LIN {X 0,Y 260.173,Z 449.996,A -85,B 0,C 180,E1 11651.487,E2 11651.487} C_VEL
LIN {X 0,Y 247.956,Z 426.22,A -85,B 0,C 180,E1 11648.205,E2 11648.205} C_VEL
LIN {X 0,Y 243.469,Z 417.822,A -85,B 0,C 180,E1 11646.84,E2 11646.84} C_VEL
LIN {X 0,Y 237.54,Z 404.393,A -85,B 0,C 180,E1 11643.464,E2 11643.464} C_VEL
LIN {X 0,Y 234.75,Z 397.683,A -85,B 0,C 180,E1 11641.737,E2 11641.737} C_VEL
LIN {X 0,Y 234.741,Z 397.554,A -85,B 0,C 180,E1 11636.558,E2 11636.558} C_VEL
LIN {X 0,Y 234.73,Z 397.556,A -85,B 0,C 180,E1 11631.489,E2 11631.489} C_VEL
LIN {X 0,Y 234.745,Z 397.554,A -85,B 0,C 180,E1 11626.327,E2 11626.327} C_VEL
LIN {X 0,Y 234.727,Z 397.561,A -85,B 0,C 180,E1 11621.3,E2 11621.3} C_VEL
LIN {X 0,Y 234.75,Z 397.558,A -85,B 0,C 180,E1 11616.113,E2 11616.113} C_VEL
LIN {X 0,Y 234.722,Z 397.559,A -85,B 0,C 180,E1 11610.976,E2 11610.976} C_VEL
LIN {X 0,Y 234.739,Z 397.555,A -85,B 0,C 180,E1 11605.847,E2 11605.847} C_VEL
LIN {X 0,Y 234.724,Z 397.557,A -85,B 0,C 180,E1 11600.685,E2 11600.685} C_VEL
LIN {X 0,Y 234.752,Z 397.559,A -85,B 0,C 180,E1 11595.698,E2 11595.698} C_VEL
LIN {X 0,Y 234.734,Z 397.56,A -85,B 0,C 180,E1 11590.282,E2 11590.282} C_VEL
LIN {X 0,Y 234.736,Z 397.556,A -85,B 0,C 180,E1 11585.327,E2 11585.327} C_VEL
LIN {X 0,Y 234.735,Z 397.557,A -85,B 0,C 180,E1 11580.108,E2 11580.108} C_VEL
LIN {X 0,Y 234.732,Z 397.564,A -85,B 0,C 180,E1 11575.195,E2 11575.195} C_VEL
LIN {X 0,Y 234.756,Z 397.673,A -85,B 0,C 180,E1 11573.699,E2 11573.699} C_VEL
LIN {X 0,Y 239.266,Z 412.086,A -85,B 0,C 180,E1 11568.68,E2 11568.68} C_VEL
LIN {X 0,Y 243.442,Z 426.646,A -85,B 0,C 180,E1 11564.048,E2 11564.048} C_VEL
LIN {X 0,Y 247.26,Z 441.444,A -85,B 0,C 180,E1 11559.711,E2 11559.711} C_VEL
LIN {X 0,Y 250.149,Z 453.996,A -85,B 0,C 180,E1 11556.269,E2 11556.269} C_VEL
LIN {X 0,Y 245.768,Z 476.519,A -85,B 0,C 180,E1 11551.382,E2 11551.382} C_VEL
LIN {X 0,Y 248.92,Z 517.799,A -85,B 0,C 180,E1 11548.969,E2 11548.969} C_VEL
LIN {X 0,Y 248.866,Z 523.548,A -85,B 0,C 180,E1 11548.677,E2 11548.677} C_VEL
LIN {X 0,Y 242.887,Z 615.376,A -85,B 0,C 180,E1 11544.277,E2 11544.277} C_VEL
LIN {X 0,Y 241.688,Z 633.773,A -85,B 0,C 180,E1 11542.949,E2 11542.949} C_VEL
LIN {X 0,Y 240.184,Z 651.793,A -85,B 0,C 180,E1 11541.173,E2 11541.173} C_VEL
LIN {X 0,Y 238.661,Z 668.194,A -85,B 0,C 180,E1 11539.074,E2 11539.074} C_VEL
LIN {X 0,Y 238.095,Z 674.333,A -85,B 0,C 180,E1 11538.142,E2 11538.142} C_VEL
LIN {X 0,Y 236.506,Z 680.701,A -85,B 0,C 180,E1 11537.118,E2 11537.118} C_VEL
LIN {X 0,Y 230.234,Z 693.25,A -85,B 0,C 180,E1 11534.856,E2 11534.856} C_VEL
LIN {X 0,Y 227.886,Z 699.683,A -85,B 0,C 180,E1 11533.431,E2 11533.431} C_VEL
LIN {X 0,Y 227.659,Z 701.248,A -85,B 0,C 180,E1 11533.044,E2 11533.044} C_VEL
LIN {X 0,Y 226.821,Z 712.8,A -85,B 0,C 180,E1 11529.9,E2 11529.9} C_VEL
LIN {X 0,Y 226.363,Z 723.238,A -85,B 0,C 180,E1 11526.34,E2 11526.34} C_VEL
LIN {X 0,Y 226.411,Z 731.344,A -85,B 0,C 180,E1 11522.785,E2 11522.785} C_VEL
LIN {X 0,Y 227.03,Z 738.033,A -85,B 0,C 180,E1 11518.991,E2 11518.991} C_VEL
LIN {X 0,Y 228.408,Z 742.937,A -85,B 0,C 180,E1 11514.978,E2 11514.978} C_VEL
LIN {X 0,Y 230.514,Z 745.783,A -85,B 0,C 180,E1 11511.268,E2 11511.268} C_VEL
LIN {X 0,Y 233.668,Z 746.873,A -85,B 0,C 180,E1 11507.395,E2 11507.395} C_VEL
LIN {X 0,Y 237.813,Z 746.163,A -85,B 0,C 180,E1 11503.639,E2 11503.639} C_VEL
LIN {X 0,Y 242.935,Z 743.576,A -85,B 0,C 180,E1 11500.025,E2 11500.025} C_VEL
LIN {X 0,Y 249.037,Z 739.206,A -85,B 0,C 180,E1 11496.58,E2 11496.58} C_VEL
LIN {X 0,Y 255.625,Z 733.401,A -85,B 0,C 180,E1 11493.519,E2 11493.519} C_VEL
LIN {X 0,Y 264.087,Z 724.771,A -85,B 0,C 180,E1 11490.266,E2 11490.266} C_VEL
LIN {X 0,Y 272.968,Z 714.412,A -85,B 0,C 180,E1 11487.422,E2 11487.422} C_VEL
LIN {X 0,Y 281.754,Z 702.992,A -85,B 0,C 180,E1 11485.06,E2 11485.06} C_VEL
LIN {X 0,Y 291.09,Z 689.414,A -85,B 0,C 180,E1 11482.928,E2 11482.928} C_VEL
LIN {X 0,Y 299.888,Z 674.728,A -85,B 0,C 180,E1 11481.185,E2 11481.185} C_VEL
LIN {X 0,Y 304.796,Z 665.496,A -85,B 0,C 180,E1 11480.292,E2 11480.292} C_VEL
LIN {X 0,Y 295.693,Z 684.166,A -85,B 0,C 180,E1 11479.091,E2 11479.091} C_VEL
LIN {X 0,Y 286.363,Z 701.007,A -85,B 0,C 180,E1 11477.602,E2 11477.602} C_VEL
LIN {X 0,Y 276.278,Z 717.417,A -85,B 0,C 180,E1 11475.624,E2 11475.624} C_VEL
LIN {X 0,Y 266.118,Z 732.842,A -85,B 0,C 180,E1 11473.142,E2 11473.142} C_VEL
LIN {X 0,Y 256.713,Z 746.406,A -85,B 0,C 180,E1 11470.282,E2 11470.282} C_VEL
LIN {X 0,Y 247.986,Z 758.698,A -85,B 0,C 180,E1 11466.924,E2 11466.924} C_VEL
LIN {X 0,Y 240.245,Z 769.768,A -85,B 0,C 180,E1 11463.039,E2 11463.039} C_VEL
LIN {X 0,Y 233.52,Z 779.982,A -85,B 0,C 180,E1 11458.377,E2 11458.377} C_VEL
LIN {X 0,Y 228.844,Z 788.193,A -85,B 0,C 180,E1 11453.428,E2 11453.428} C_VEL
LIN {X 0,Y 226.352,Z 794.238,A -85,B 0,C 180,E1 11448.545,E2 11448.545} C_VEL
LIN {X 0,Y 225.176,Z 804.136,A -85,B 0,C 180,E1 11444.398,E2 11444.398} C_VEL
LIN {X 0,Y 224.691,Z 811.895,A -85,B 0,C 180,E1 11440.253,E2 11440.253} C_VEL
LIN {X 0,Y 224.74,Z 817.761,A -85,B 0,C 180,E1 11436.13,E2 11436.13} C_VEL
LIN {X 0,Y 224.855,Z 821.641,A -85,B 0,C 180,E1 11432.294,E2 11432.294} C_VEL
LIN {X 0,Y 224.745,Z 823.926,A -85,B 0,C 180,E1 11428.725,E2 11428.725} C_VEL
LIN {X 0,Y 224.369,Z 825.073,A -85,B 0,C 180,E1 11424.63,E2 11424.63} C_VEL
LIN {X 0,Y 224.279,Z 824.752,A -85,B 0,C 180,E1 11419.987,E2 11419.987} C_VEL
LIN {X 0,Y 225.314,Z 822.532,A -85,B 0,C 180,E1 11414.822,E2 11414.822} C_VEL
LIN {X 0,Y 228.103,Z 818.227,A -85,B 0,C 180,E1 11409.472,E2 11409.472} C_VEL
LIN {X 0,Y 232.879,Z 811.96,A -85,B 0,C 180,E1 11404.301,E2 11404.301} C_VEL
LIN {X 0,Y 239.69,Z 803.753,A -85,B 0,C 180,E1 11399.408,E2 11399.408} C_VEL
LIN {X 0,Y 248.538,Z 793.638,A -85,B 0,C 180,E1 11394.88,E2 11394.88} C_VEL
LIN {X 0,Y 259.353,Z 781.523,A -85,B 0,C 180,E1 11390.783,E2 11390.783} C_VEL
LIN {X 0,Y 271.422,Z 768.109,A -85,B 0,C 180,E1 11387.327,E2 11387.327} C_VEL
LIN {X 0,Y 284.436,Z 753.541,A -85,B 0,C 180,E1 11384.472,E2 11384.472} C_VEL
LIN {X 0,Y 288.888,Z 748.523,A -85,B 0,C 180,E1 11383.627,E2 11383.627} C_VEL
LIN {X 0,Y 276.067,Z 761.536,A -85,B 0,C 180,E1 11380.687,E2 11380.687} C_VEL
LIN {X 0,Y 264.26,Z 772.98,A -85,B 0,C 180,E1 11377.256,E2 11377.256} C_VEL
LIN {X 0,Y 253.496,Z 782.998,A -85,B 0,C 180,E1 11373.247,E2 11373.247} C_VEL
LIN {X 0,Y 244.427,Z 790.978,A -85,B 0,C 180,E1 11368.861,E2 11368.861} C_VEL
LIN {X 0,Y 237.116,Z 796.985,A -85,B 0,C 180,E1 11364.143,E2 11364.143} C_VEL
LIN {X 0,Y 231.58,Z 801.07,A -85,B 0,C 180,E1 11359.155,E2 11359.155} C_VEL
LIN {X 0,Y 227.872,Z 803.179,A -85,B 0,C 180,E1 11354.137,E2 11354.137} C_VEL
LIN {X 0,Y 225.685,Z 803.454,A -85,B 0,C 180,E1 11349.177,E2 11349.177} C_VEL
LIN {X 0,Y 224.64,Z 801.992,A -85,B 0,C 180,E1 11344.339,E2 11344.339} C_VEL
LIN {X 0,Y 224.296,Z 798.959,A -85,B 0,C 180,E1 11339.744,E2 11339.744} C_VEL
LIN {X 0,Y 224.27,Z 794.49,A -85,B 0,C 180,E1 11335.397,E2 11335.397} C_VEL
LIN {X 0,Y 224.606,Z 788.308,A -85,B 0,C 180,E1 11331.036,E2 11331.036} C_VEL
LIN {X 0,Y 225.458,Z 780.224,A -85,B 0,C 180,E1 11326.667,E2 11326.667} C_VEL
LIN {X 0,Y 226.903,Z 770.573,A -85,B 0,C 180,E1 11322.563,E2 11322.563} C_VEL
LIN {X 0,Y 228.921,Z 759.495,A -85,B 0,C 180,E1 11318.745,E2 11318.745} C_VEL
LIN {X 0,Y 231.574,Z 746.383,A -85,B 0,C 180,E1 11315.055,E2 11315.055} C_VEL
LIN {X 0,Y 234.709,Z 731.505,A -85,B 0,C 180,E1 11311.641,E2 11311.641} C_VEL
LIN {X 0,Y 238.092,Z 715.357,A -85,B 0,C 180,E1 11308.618,E2 11308.618} C_VEL
LIN {X 0,Y 241.496,Z 698.159,A -85,B 0,C 180,E1 11306.017,E2 11306.017} C_VEL
LIN {X 0,Y 244.946,Z 679.052,A -85,B 0,C 180,E1 11303.709,E2 11303.709} C_VEL
LIN {X 0,Y 247.939,Z 660.023,A -85,B 0,C 180,E1 11301.902,E2 11301.902} C_VEL
LIN {X 0,Y 250.598,Z 639.472,A -85,B 0,C 180,E1 11300.42,E2 11300.42} C_VEL
LIN {X 0,Y 252.79,Z 617.241,A -85,B 0,C 180,E1 11299.297,E2 11299.297} C_VEL
LIN {X 0,Y 265.525,Z 478.492,A -85,B 0,C 180,E1 11293.746,E2 11293.746} C_VEL
LIN {X 0,Y 253.283,Z 452.497,A -85,B 0,C 180,E1 11290.57,E2 11290.57} C_VEL
LIN {X 0,Y 241.211,Z 429.066,A -85,B 0,C 180,E1 11287.206,E2 11287.206} C_VEL
LIN {X 0,Y 235.673,Z 418.905,A -85,B 0,C 180,E1 11285.538,E2 11285.538} C_VEL
LIN {X 0,Y 229.773,Z 405.644,A -85,B 0,C 180,E1 11282.065,E2 11282.065} C_VEL
LIN {X 0,Y 226.886,Z 399.007,A -85,B 0,C 180,E1 11280.259,E2 11280.259} C_VEL
LIN {X 0,Y 226.808,Z 398.546,A -85,B 0,C 180,E1 11280.046,E2 11280.046} C_VEL
LIN {X 0,Y 226.797,Z 398.546,A -85,B 0,C 180,E1 11274.745,E2 11274.745} C_VEL
LIN {X 0,Y 226.802,Z 398.544,A -85,B 0,C 180,E1 11269.844,E2 11269.844} C_VEL
LIN {X 0,Y 226.809,Z 398.544,A -85,B 0,C 180,E1 11264.292,E2 11264.292} C_VEL
LIN {X 0,Y 226.785,Z 398.54,A -85,B 0,C 180,E1 11259.036,E2 11259.036} C_VEL
LIN {X 0,Y 226.799,Z 398.536,A -85,B 0,C 180,E1 11254.045,E2 11254.045} C_VEL
LIN {X 0,Y 226.786,Z 398.537,A -85,B 0,C 180,E1 11248.737,E2 11248.737} C_VEL
LIN {X 0,Y 226.803,Z 398.541,A -85,B 0,C 180,E1 11243.672,E2 11243.672} C_VEL
LIN {X 0,Y 226.797,Z 398.543,A -85,B 0,C 180,E1 11238.158,E2 11238.158} C_VEL
LIN {X 0,Y 226.789,Z 398.544,A -85,B 0,C 180,E1 11233.079,E2 11233.079} C_VEL
LIN {X 0,Y 226.819,Z 398.547,A -85,B 0,C 180,E1 11227.722,E2 11227.722} C_VEL
LIN {X 0,Y 226.791,Z 398.546,A -85,B 0,C 180,E1 11222.395,E2 11222.395} C_VEL
LIN {X 0,Y 226.799,Z 398.551,A -85,B 0,C 180,E1 11217.357,E2 11217.357} C_VEL
LIN {X 0,Y 226.816,Z 398.762,A -85,B 0,C 180,E1 11214.958,E2 11214.958} C_VEL
LIN {X 0,Y 230.994,Z 411.865,A -85,B 0,C 180,E1 11210.162,E2 11210.162} C_VEL
LIN {X 0,Y 235.121,Z 426.023,A -85,B 0,C 180,E1 11205.439,E2 11205.439} C_VEL
LIN {X 0,Y 239.156,Z 441.502,A -85,B 0,C 180,E1 11200.708,E2 11200.708} C_VEL
LIN {X 0,Y 242.421,Z 455.848,A -85,B 0,C 180,E1 11196.657,E2 11196.657} C_VEL
LIN {X 0,Y 238.264,Z 476.263,A -85,B 0,C 180,E1 11192.093,E2 11192.093} C_VEL
LIN {X 0,Y 241.022,Z 515.382,A -85,B 0,C 180,E1 11189.736,E2 11189.736} C_VEL
LIN {X 0,Y 241.375,Z 522.415,A -85,B 0,C 180,E1 11189.33,E2 11189.33} C_VEL
LIN {X 0,Y 235.056,Z 615.529,A -85,B 0,C 180,E1 11184.671,E2 11184.671} C_VEL
LIN {X 0,Y 233.819,Z 634.044,A -85,B 0,C 180,E1 11183.301,E2 11183.301} C_VEL
LIN {X 0,Y 232.267,Z 652.222,A -85,B 0,C 180,E1 11181.464,E2 11181.464} C_VEL
LIN {X 0,Y 230.669,Z 669.136,A -85,B 0,C 180,E1 11179.235,E2 11179.235} C_VEL
LIN {X 0,Y 229.234,Z 684.132,A -85,B 0,C 180,E1 11176.731,E2 11176.731} C_VEL
LIN {X 0,Y 227.894,Z 698.526,A -85,B 0,C 180,E1 11173.705,E2 11173.705} C_VEL
LIN {X 0,Y 227.659,Z 701.248,A -85,B 0,C 180,E1 11173.044,E2 11173.044} C_VEL
LIN {X 0,Y 226.241,Z 706.651,A -85,B 0,C 180,E1 11171.674,E2 11171.674} C_VEL
LIN {X 0,Y 221.199,Z 715.74,A -85,B 0,C 180,E1 11169.06,E2 11169.06} C_VEL
LIN {X 0,Y 218.61,Z 721.607,A -85,B 0,C 180,E1 11167.039,E2 11167.039} C_VEL
LIN {X 0,Y 218.362,Z 723.457,A -85,B 0,C 180,E1 11166.321,E2 11166.321} C_VEL
LIN {X 0,Y 218.429,Z 731.929,A -85,B 0,C 180,E1 11162.624,E2 11162.624} C_VEL
LIN {X 0,Y 219.104,Z 738.783,A -85,B 0,C 180,E1 11158.693,E2 11158.693} C_VEL
LIN {X 0,Y 220.481,Z 743.749,A -85,B 0,C 180,E1 11154.797,E2 11154.797} C_VEL
LIN {X 0,Y 222.868,Z 747.071,A -85,B 0,C 180,E1 11150.706,E2 11150.706} C_VEL
LIN {X 0,Y 226.029,Z 748.493,A -85,B 0,C 180,E1 11146.962,E2 11146.962} C_VEL
LIN {X 0,Y 230.388,Z 748.169,A -85,B 0,C 180,E1 11143.096,E2 11143.096} C_VEL
LIN {X 0,Y 236.173,Z 745.942,A -85,B 0,C 180,E1 11139.169,E2 11139.169} C_VEL
LIN {X 0,Y 243.076,Z 741.661,A -85,B 0,C 180,E1 11135.453,E2 11135.453} C_VEL
LIN {X 0,Y 250.606,Z 735.843,A -85,B 0,C 180,E1 11132.173,E2 11132.173} C_VEL
LIN {X 0,Y 259.619,Z 727.558,A -85,B 0,C 180,E1 11128.931,E2 11128.931} C_VEL
LIN {X 0,Y 269.058,Z 717.724,A -85,B 0,C 180,E1 11126.123,E2 11126.123} C_VEL
LIN {X 0,Y 278.736,Z 706.354,A -85,B 0,C 180,E1 11123.71,E2 11123.71} C_VEL
LIN {X 0,Y 288.483,Z 693.497,A -85,B 0,C 180,E1 11121.655,E2 11121.655} C_VEL
LIN {X 0,Y 293.944,Z 685.526,A -85,B 0,C 180,E1 11120.589,E2 11120.589} C_VEL
LIN {X 0,Y 283.738,Z 702.351,A -85,B 0,C 180,E1 11119.102,E2 11119.102} C_VEL
LIN {X 0,Y 272.862,Z 718.607,A -85,B 0,C 180,E1 11117.128,E2 11117.128} C_VEL
LIN {X 0,Y 261.868,Z 733.698,A -85,B 0,C 180,E1 11114.632,E2 11114.632} C_VEL
LIN {X 0,Y 251.377,Z 747.383,A -85,B 0,C 180,E1 11111.625,E2 11111.625} C_VEL
LIN {X 0,Y 241.685,Z 759.768,A -85,B 0,C 180,E1 11108.055,E2 11108.055} C_VEL
LIN {X 0,Y 233.123,Z 770.752,A -85,B 0,C 180,E1 11103.888,E2 11103.888} C_VEL
LIN {X 0,Y 226.07,Z 780.267,A -85,B 0,C 180,E1 11099.112,E2 11099.112} C_VEL
LIN {X 0,Y 221.134,Z 787.904,A -85,B 0,C 180,E1 11094.013,E2 11094.013} C_VEL
LIN {X 0,Y 218.389,Z 793.726,A -85,B 0,C 180,E1 11088.692,E2 11088.692} C_VEL
LIN {X 0,Y 218.124,Z 795.391,A -85,B 0,C 180,E1 11087.886,E2 11087.886} C_VEL
LIN {X 0,Y 217.123,Z 804.41,A -85,B 0,C 180,E1 11083.855,E2 11083.855} C_VEL
LIN {X 0,Y 216.731,Z 811.969,A -85,B 0,C 180,E1 11079.56,E2 11079.56} C_VEL
LIN {X 0,Y 216.827,Z 817.331,A -85,B 0,C 180,E1 11075.557,E2 11075.557} C_VEL
LIN {X 0,Y 216.931,Z 821.127,A -85,B 0,C 180,E1 11071.585,E2 11071.585} C_VEL
LIN {X 0,Y 216.724,Z 823.337,A -85,B 0,C 180,E1 11067.885,E2 11067.885} C_VEL
LIN {X 0,Y 216.327,Z 824.428,A -85,B 0,C 180,E1 11063.577,E2 11063.577} C_VEL
LIN {X 0,Y 216.424,Z 824.012,A -85,B 0,C 180,E1 11058.542,E2 11058.542} C_VEL
LIN {X 0,Y 217.907,Z 821.738,A -85,B 0,C 180,E1 11053.197,E2 11053.197} C_VEL
LIN {X 0,Y 221.335,Z 817.444,A -85,B 0,C 180,E1 11047.7,E2 11047.7} C_VEL
LIN {X 0,Y 226.871,Z 811.272,A -85,B 0,C 180,E1 11042.435,E2 11042.435} C_VEL
LIN {X 0,Y 234.507,Z 803.265,A -85,B 0,C 180,E1 11037.505,E2 11037.505} C_VEL
LIN {X 0,Y 244.496,Z 793.175,A -85,B 0,C 180,E1 11032.887,E2 11032.887} C_VEL
LIN {X 0,Y 256.497,Z 781.234,A -85,B 0,C 180,E1 11028.792,E2 11028.792} C_VEL
LIN {X 0,Y 269.439,Z 768.323,A -85,B 0,C 180,E1 11025.464,E2 11025.464} C_VEL
LIN {X 0,Y 278.882,Z 758.747,A -85,B 0,C 180,E1 11023.501,E2 11023.501} C_VEL
LIN {X 0,Y 265.731,Z 770.475,A -85,B 0,C 180,E1 11020.329,E2 11020.329} C_VEL
LIN {X 0,Y 254.057,Z 780.398,A -85,B 0,C 180,E1 11016.741,E2 11016.741} C_VEL
LIN {X 0,Y 243.428,Z 788.893,A -85,B 0,C 180,E1 11012.552,E2 11012.552} C_VEL
LIN {X 0,Y 234.569,Z 795.523,A -85,B 0,C 180,E1 11007.961,E2 11007.961} C_VEL
LIN {X 0,Y 227.535,Z 800.312,A -85,B 0,C 180,E1 11003.022,E2 11003.022} C_VEL
LIN {X 0,Y 222.551,Z 803.132,A -85,B 0,C 180,E1 10998.059,E2 10998.059} C_VEL
LIN {X 0,Y 219.181,Z 804.232,A -85,B 0,C 180,E1 10992.916,E2 10992.916} C_VEL
LIN {X 0,Y 217.323,Z 803.605,A -85,B 0,C 180,E1 10987.933,E2 10987.933} C_VEL
LIN {X 0,Y 216.5,Z 801.443,A -85,B 0,C 180,E1 10983.177,E2 10983.177} C_VEL
LIN {X 0,Y 216.257,Z 797.906,A -85,B 0,C 180,E1 10978.675,E2 10978.675} C_VEL
LIN {X 0,Y 216.327,Z 792.777,A -85,B 0,C 180,E1 10974.164,E2 10974.164} C_VEL
LIN {X 0,Y 216.805,Z 785.867,A -85,B 0,C 180,E1 10969.638,E2 10969.638} C_VEL
LIN {X 0,Y 217.817,Z 777.523,A -85,B 0,C 180,E1 10965.376,E2 10965.376} C_VEL
LIN {X 0,Y 219.516,Z 767.158,A -85,B 0,C 180,E1 10961.131,E2 10961.131} C_VEL
LIN {X 0,Y 221.825,Z 755.285,A -85,B 0,C 180,E1 10957.192,E2 10957.192} C_VEL
LIN {X 0,Y 224.658,Z 741.873,A -85,B 0,C 180,E1 10953.572,E2 10953.572} C_VEL
LIN {X 0,Y 228.015,Z 726.348,A -85,B 0,C 180,E1 10950.151,E2 10950.151} C_VEL
LIN {X 0,Y 231.524,Z 709.781,A -85,B 0,C 180,E1 10947.181,E2 10947.181} C_VEL
LIN {X 0,Y 235.001,Z 692.323,A -85,B 0,C 180,E1 10944.645,E2 10944.645} C_VEL
LIN {X 0,Y 238.291,Z 673.952,A -85,B 0,C 180,E1 10942.525,E2 10942.525} C_VEL
LIN {X 0,Y 241.304,Z 654.325,A -85,B 0,C 180,E1 10940.755,E2 10940.755} C_VEL
LIN {X 0,Y 243.946,Z 633.235,A -85,B 0,C 180,E1 10939.33,E2 10939.33} C_VEL
LIN {X 0,Y 246.955,Z 600.782,A -85,B 0,C 180,E1 10937.83,E2 10937.83} C_VEL
LIN {X 0,Y 258.526,Z 480.835,A -85,B 0,C 180,E1 10932.898,E2 10932.898} C_VEL
LIN {X 0,Y 246.755,Z 455.798,A -85,B 0,C 180,E1 10929.733,E2 10929.733} C_VEL
LIN {X 0,Y 234.648,Z 432.136,A -85,B 0,C 180,E1 10926.207,E2 10926.207} C_VEL
LIN {X 0,Y 227.524,Z 419.019,A -85,B 0,C 180,E1 10923.925,E2 10923.925} C_VEL
LIN {X 0,Y 221.6,Z 406.138,A -85,B 0,C 180,E1 10920.354,E2 10920.354} C_VEL
LIN {X 0,Y 220.029,Z 402.826,A -85,B 0,C 180,E1 10919.392,E2 10919.392} C_VEL
LIN {X 0,Y 218.871,Z 399.536,A -85,B 0,C 180,E1 10918.436,E2 10918.436} C_VEL
LIN {X 0,Y 218.849,Z 399.534,A -85,B 0,C 180,E1 10913.136,E2 10913.136} C_VEL
LIN {X 0,Y 218.861,Z 399.531,A -85,B 0,C 180,E1 10907.824,E2 10907.824} C_VEL
LIN {X 0,Y 218.858,Z 399.53,A -85,B 0,C 180,E1 10902.399,E2 10902.399} C_VEL
LIN {X 0,Y 218.848,Z 399.536,A -85,B 0,C 180,E1 10897.086,E2 10897.086} C_VEL
LIN {X 0,Y 218.861,Z 399.533,A -85,B 0,C 180,E1 10891.833,E2 10891.833} C_VEL
LIN {X 0,Y 218.853,Z 399.53,A -85,B 0,C 180,E1 10886.333,E2 10886.333} C_VEL
LIN {X 0,Y 218.847,Z 399.533,A -85,B 0,C 180,E1 10881.064,E2 10881.064} C_VEL
LIN {X 0,Y 218.874,Z 399.536,A -85,B 0,C 180,E1 10875.719,E2 10875.719} C_VEL
LIN {X 0,Y 218.856,Z 399.537,A -85,B 0,C 180,E1 10870.24,E2 10870.24} C_VEL
LIN {X 0,Y 218.854,Z 399.535,A -85,B 0,C 180,E1 10865.145,E2 10865.145} C_VEL
LIN {X 0,Y 218.873,Z 399.535,A -85,B 0,C 180,E1 10859.7,E2 10859.7} C_VEL
LIN {X 0,Y 218.857,Z 399.606,A -85,B 0,C 180,E1 10856.36,E2 10856.36} C_VEL
LIN {X 0,Y 223.202,Z 413.233,A -85,B 0,C 180,E1 10851.16,E2 10851.16} C_VEL
LIN {X 0,Y 227.144,Z 426.794,A -85,B 0,C 180,E1 10846.457,E2 10846.457} C_VEL
LIN {X 0,Y 230.818,Z 440.709,A -85,B 0,C 180,E1 10842.02,E2 10842.02} C_VEL
LIN {X 0,Y 234.582,Z 456.632,A -85,B 0,C 180,E1 10837.332,E2 10837.332} C_VEL
LIN {X 0,Y 234.448,Z 458.68,A -85,B 0,C 180,E1 10836.818,E2 10836.818} C_VEL
LIN {X 0,Y 230.763,Z 476.253,A -85,B 0,C 180,E1 10832.806,E2 10832.806} C_VEL
LIN {X 0,Y 233.15,Z 513.277,A -85,B 0,C 180,E1 10830.493,E2 10830.493} C_VEL
LIN {X 0,Y 233.739,Z 522.892,A -85,B 0,C 180,E1 10829.909,E2 10829.909} C_VEL
LIN {X 0,Y 227.192,Z 616.395,A -85,B 0,C 180,E1 10825.044,E2 10825.044} C_VEL
LIN {X 0,Y 225.927,Z 634.74,A -85,B 0,C 180,E1 10823.637,E2 10823.637} C_VEL
LIN {X 0,Y 224.411,Z 652.021,A -85,B 0,C 180,E1 10821.841,E2 10821.841} C_VEL
LIN {X 0,Y 222.678,Z 669.852,A -85,B 0,C 180,E1 10819.407,E2 10819.407} C_VEL
LIN {X 0,Y 221.143,Z 685.516,A -85,B 0,C 180,E1 10816.685,E2 10816.685} C_VEL
LIN {X 0,Y 219.757,Z 700.453,A -85,B 0,C 180,E1 10813.418,E2 10813.418} C_VEL
LIN {X 0,Y 218.831,Z 712.873,A -85,B 0,C 180,E1 10809.999,E2 10809.999} C_VEL
LIN {X 0,Y 218.37,Z 723.019,A -85,B 0,C 180,E1 10806.49,E2 10806.49} C_VEL
LIN {X 0,Y 218.362,Z 723.457,A -85,B 0,C 180,E1 10806.321,E2 10806.321} C_VEL
LIN {X 0,Y 217.338,Z 727.654,A -85,B 0,C 180,E1 10804.624,E2 10804.624} C_VEL
LIN {X 0,Y 213.122,Z 734.447,A -85,B 0,C 180,E1 10801.383,E2 10801.383} C_VEL
LIN {X 0,Y 211.234,Z 738.621,A -85,B 0,C 180,E1 10798.957,E2 10798.957} C_VEL
LIN {X 0,Y 211.246,Z 739.885,A -85,B 0,C 180,E1 10798.12,E2 10798.12} C_VEL
LIN {X 0,Y 212.805,Z 745.021,A -85,B 0,C 180,E1 10794.067,E2 10794.067} C_VEL
LIN {X 0,Y 215.434,Z 748.498,A -85,B 0,C 180,E1 10789.842,E2 10789.842} C_VEL
LIN {X 0,Y 219.161,Z 750.158,A -85,B 0,C 180,E1 10785.738,E2 10785.738} C_VEL
LIN {X 0,Y 223.961,Z 749.962,A -85,B 0,C 180,E1 10781.79,E2 10781.79} C_VEL
LIN {X 0,Y 230.251,Z 747.901,A -85,B 0,C 180,E1 10777.803,E2 10777.803} C_VEL
LIN {X 0,Y 237.239,Z 744.185,A -85,B 0,C 180,E1 10774.272,E2 10774.272} C_VEL
LIN {X 0,Y 246.303,Z 737.959,A -85,B 0,C 180,E1 10770.581,E2 10770.581} C_VEL
LIN {X 0,Y 255.954,Z 729.961,A -85,B 0,C 180,E1 10767.379,E2 10767.379} C_VEL
LIN {X 0,Y 266.006,Z 720.521,A -85,B 0,C 180,E1 10764.63,E2 10764.63} C_VEL
LIN {X 0,Y 276.939,Z 708.776,A -85,B 0,C 180,E1 10762.138,E2 10762.138} C_VEL
LIN {X 0,Y 283.13,Z 701.492,A -85,B 0,C 180,E1 10760.869,E2 10760.869} C_VEL
LIN {X 0,Y 272.701,Z 715.955,A -85,B 0,C 180,E1 10759.212,E2 10759.212} C_VEL
LIN {X 0,Y 261.298,Z 730.518,A -85,B 0,C 180,E1 10756.959,E2 10756.959} C_VEL
LIN {X 0,Y 249.291,Z 744.892,A -85,B 0,C 180,E1 10753.938,E2 10753.938} C_VEL
LIN {X 0,Y 238.691,Z 757.117,A -85,B 0,C 180,E1 10750.488,E2 10750.488} C_VEL
LIN {X 0,Y 229.127,Z 768.075,A -85,B 0,C 180,E1 10746.404,E2 10746.404} C_VEL
LIN {X 0,Y 221,Z 777.6,A -85,B 0,C 180,E1 10741.656,E2 10741.656} C_VEL
LIN {X 0,Y 214.779,Z 785.642,A -85,B 0,C 180,E1 10736.248,E2 10736.248} C_VEL
LIN {X 0,Y 211.012,Z 791.778,A -85,B 0,C 180,E1 10730.527,E2 10730.527} C_VEL
LIN {X 0,Y 210.285,Z 793.753,A -85,B 0,C 180,E1 10728.289,E2 10728.289} C_VEL
LIN {X 0,Y 209.173,Z 803.519,A -85,B 0,C 180,E1 10723.828,E2 10723.828} C_VEL
LIN {X 0,Y 208.796,Z 811.138,A -85,B 0,C 180,E1 10719.37,E2 10719.37} C_VEL
LIN {X 0,Y 208.917,Z 816.548,A -85,B 0,C 180,E1 10715.217,E2 10715.217} C_VEL
LIN {X 0,Y 209.003,Z 820.383,A -85,B 0,C 180,E1 10711.097,E2 10711.097} C_VEL
LIN {X 0,Y 208.722,Z 822.582,A -85,B 0,C 180,E1 10707.254,E2 10707.254} C_VEL
LIN {X 0,Y 208.309,Z 823.749,A -85,B 0,C 180,E1 10702.554,E2 10702.554} C_VEL
LIN {X 0,Y 208.681,Z 823.271,A -85,B 0,C 180,E1 10696.986,E2 10696.986} C_VEL
LIN {X 0,Y 210.826,Z 820.814,A -85,B 0,C 180,E1 10691.186,E2 10691.186} C_VEL
LIN {X 0,Y 215.066,Z 816.488,A -85,B 0,C 180,E1 10685.558,E2 10685.558} C_VEL
LIN {X 0,Y 221.507,Z 810.365,A -85,B 0,C 180,E1 10680.229,E2 10680.229} C_VEL
LIN {X 0,Y 230.572,Z 802.107,A -85,B 0,C 180,E1 10675.081,E2 10675.081} C_VEL
LIN {X 0,Y 241.906,Z 791.995,A -85,B 0,C 180,E1 10670.467,E2 10670.467} C_VEL
LIN {X 0,Y 254.707,Z 780.611,A -85,B 0,C 180,E1 10666.609,E2 10666.609} C_VEL
LIN {X 0,Y 268.804,Z 767.938,A -85,B 0,C 180,E1 10663.373,E2 10663.373} C_VEL
LIN {X 0,Y 255.316,Z 778.381,A -85,B 0,C 180,E1 10659.96,E2 10659.96} C_VEL
LIN {X 0,Y 242.685,Z 787.603,A -85,B 0,C 180,E1 10655.805,E2 10655.805} C_VEL
LIN {X 0,Y 232.414,Z 794.609,A -85,B 0,C 180,E1 10651.369,E2 10651.369} C_VEL
LIN {X 0,Y 223.626,Z 800.049,A -85,B 0,C 180,E1 10646.272,E2 10646.272} C_VEL
LIN {X 0,Y 217.175,Z 803.362,A -85,B 0,C 180,E1 10641.045,E2 10641.045} C_VEL
LIN {X 0,Y 212.635,Z 804.846,A -85,B 0,C 180,E1 10635.547,E2 10635.547} C_VEL
LIN {X 0,Y 209.975,Z 804.504,A -85,B 0,C 180,E1 10630.147,E2 10630.147} C_VEL
LIN {X 0,Y 208.686,Z 802.38,A -85,B 0,C 180,E1 10624.74,E2 10624.74} C_VEL
LIN {X 0,Y 208.295,Z 798.734,A -85,B 0,C 180,E1 10619.725,E2 10619.725} C_VEL
LIN {X 0,Y 208.287,Z 793.714,A -85,B 0,C 180,E1 10615.043,E2 10615.043} C_VEL
LIN {X 0,Y 208.695,Z 786.931,A -85,B 0,C 180,E1 10610.346,E2 10610.346} C_VEL
LIN {X 0,Y 209.629,Z 778.731,A -85,B 0,C 180,E1 10605.921,E2 10605.921} C_VEL
LIN {X 0,Y 211.274,Z 768.528,A -85,B 0,C 180,E1 10601.513,E2 10601.513} C_VEL
LIN {X 0,Y 213.552,Z 756.84,A -85,B 0,C 180,E1 10597.422,E2 10597.422} C_VEL
LIN {X 0,Y 216.493,Z 743.187,A -85,B 0,C 180,E1 10593.533,E2 10593.533} C_VEL
LIN {X 0,Y 219.898,Z 727.832,A -85,B 0,C 180,E1 10589.989,E2 10589.989} C_VEL
LIN {X 0,Y 223.643,Z 710.655,A -85,B 0,C 180,E1 10586.776,E2 10586.776} C_VEL
LIN {X 0,Y 227.383,Z 692.388,A -85,B 0,C 180,E1 10584.037,E2 10584.037} C_VEL
LIN {X 0,Y 230.948,Z 672.931,A -85,B 0,C 180,E1 10581.749,E2 10581.749} C_VEL
LIN {X 0,Y 234.193,Z 652.141,A -85,B 0,C 180,E1 10579.858,E2 10579.858} C_VEL
LIN {X 0,Y 236.818,Z 631.335,A -85,B 0,C 180,E1 10578.46,E2 10578.46} C_VEL
LIN {X 0,Y 248.312,Z 515.301,A -85,B 0,C 180,E1 10573.359,E2 10573.359} C_VEL
LIN {X 0,Y 251.612,Z 483.289,A -85,B 0,C 180,E1 10572.036,E2 10572.036} C_VEL
LIN {X 0,Y 239.198,Z 456.934,A -85,B 0,C 180,E1 10568.561,E2 10568.561} C_VEL
LIN {X 0,Y 227.201,Z 433.566,A -85,B 0,C 180,E1 10564.897,E2 10564.897} C_VEL
LIN {X 0,Y 219.368,Z 419.263,A -85,B 0,C 180,E1 10562.227,E2 10562.227} C_VEL
LIN {X 0,Y 213.856,Z 407.466,A -85,B 0,C 180,E1 10558.788,E2 10558.788} C_VEL
LIN {X 0,Y 212.326,Z 404.15,A -85,B 0,C 180,E1 10557.788,E2 10557.788} C_VEL
LIN {X 0,Y 210.936,Z 400.655,A -85,B 0,C 180,E1 10556.764,E2 10556.764} C_VEL
LIN {X 0,Y 210.912,Z 400.522,A -85,B 0,C 180,E1 10551.409,E2 10551.409} C_VEL
LIN {X 0,Y 210.925,Z 400.523,A -85,B 0,C 180,E1 10545.959,E2 10545.959} C_VEL
LIN {X 0,Y 210.92,Z 400.526,A -85,B 0,C 180,E1 10540.378,E2 10540.378} C_VEL
LIN {X 0,Y 210.908,Z 400.523,A -85,B 0,C 180,E1 10535.168,E2 10535.168} C_VEL
LIN {X 0,Y 210.926,Z 400.519,A -85,B 0,C 180,E1 10529.728,E2 10529.728} C_VEL
LIN {X 0,Y 210.926,Z 400.521,A -85,B 0,C 180,E1 10524.014,E2 10524.014} C_VEL
LIN {X 0,Y 210.911,Z 400.524,A -85,B 0,C 180,E1 10518.515,E2 10518.515} C_VEL
LIN {X 0,Y 210.914,Z 400.521,A -85,B 0,C 180,E1 10513.191,E2 10513.191} C_VEL
LIN {X 0,Y 210.932,Z 400.526,A -85,B 0,C 180,E1 10507.57,E2 10507.57} C_VEL
LIN {X 0,Y 210.933,Z 400.525,A -85,B 0,C 180,E1 10501.846,E2 10501.846} C_VEL
LIN {X 0,Y 210.924,Z 400.536,A -85,B 0,C 180,E1 10497.831,E2 10497.831} C_VEL
LIN {X 0,Y 215.188,Z 413.819,A -85,B 0,C 180,E1 10492.505,E2 10492.505} C_VEL
LIN {X 0,Y 219.209,Z 427.506,A -85,B 0,C 180,E1 10487.541,E2 10487.541} C_VEL
LIN {X 0,Y 223.158,Z 442.522,A -85,B 0,C 180,E1 10482.576,E2 10482.576} C_VEL
LIN {X 0,Y 226.841,Z 458.303,A -85,B 0,C 180,E1 10477.784,E2 10477.784} C_VEL
LIN {X 0,Y 226.782,Z 460.082,A -85,B 0,C 180,E1 10477.317,E2 10477.317} C_VEL
LIN {X 0,Y 223.286,Z 476.185,A -85,B 0,C 180,E1 10473.562,E2 10473.562} C_VEL
LIN {X 0,Y 225.338,Z 511.406,A -85,B 0,C 180,E1 10471.284,E2 10471.284} C_VEL
LIN {X 0,Y 226.115,Z 523.295,A -85,B 0,C 180,E1 10470.52,E2 10470.52} C_VEL
LIN {X 0,Y 219.386,Z 616.118,A -85,B 0,C 180,E1 10465.494,E2 10465.494} C_VEL
LIN {X 0,Y 218.004,Z 635.444,A -85,B 0,C 180,E1 10463.95,E2 10463.95} C_VEL
LIN {X 0,Y 216.361,Z 653.52,A -85,B 0,C 180,E1 10461.983,E2 10461.983} C_VEL
LIN {X 0,Y 214.691,Z 670.447,A -85,B 0,C 180,E1 10459.592,E2 10459.592} C_VEL
LIN {X 0,Y 213.118,Z 686.225,A -85,B 0,C 180,E1 10456.77,E2 10456.77} C_VEL
LIN {X 0,Y 211.806,Z 700.074,A -85,B 0,C 180,E1 10453.653,E2 10453.653} C_VEL
LIN {X 0,Y 210.897,Z 711.872,A -85,B 0,C 180,E1 10450.379,E2 10450.379} C_VEL
LIN {X 0,Y 210.378,Z 722.855,A -85,B 0,C 180,E1 10446.629,E2 10446.629} C_VEL
LIN {X 0,Y 210.397,Z 731.248,A -85,B 0,C 180,E1 10442.997,E2 10442.997} C_VEL
LIN {X 0,Y 211.039,Z 738.691,A -85,B 0,C 180,E1 10438.914,E2 10438.914} C_VEL
LIN {X 0,Y 211.246,Z 739.885,A -85,B 0,C 180,E1 10438.12,E2 10438.12} C_VEL
LIN {X 0,Y 210.89,Z 742.716,A -85,B 0,C 180,E1 10436.158,E2 10436.158} C_VEL
LIN {X 0,Y 208.025,Z 747.369,A -85,B 0,C 180,E1 10432.137,E2 10432.137} C_VEL
LIN {X 0,Y 207.62,Z 749.363,A -85,B 0,C 180,E1 10429.743,E2 10429.743} C_VEL
LIN {X 0,Y 208.113,Z 749.95,A -85,B 0,C 180,E1 10428.85,E2 10428.85} C_VEL
LIN {X 0,Y 212.414,Z 751.831,A -85,B 0,C 180,E1 10424.437,E2 10424.437} C_VEL
LIN {X 0,Y 217.679,Z 751.797,A -85,B 0,C 180,E1 10420.409,E2 10420.409} C_VEL
LIN {X 0,Y 224.495,Z 749.912,A -85,B 0,C 180,E1 10416.369,E2 10416.369} C_VEL
LIN {X 0,Y 232.021,Z 746.478,A -85,B 0,C 180,E1 10412.82,E2 10412.82} C_VEL
LIN {X 0,Y 241.114,Z 740.955,A -85,B 0,C 180,E1 10409.332,E2 10409.332} C_VEL
LIN {X 0,Y 251.303,Z 733.551,A -85,B 0,C 180,E1 10406.15,E2 10406.15} C_VEL
LIN {X 0,Y 262.508,Z 724.076,A -85,B 0,C 180,E1 10403.274,E2 10403.274} C_VEL
LIN {X 0,Y 272.36,Z 714.691,A -85,B 0,C 180,E1 10401.145,E2 10401.145} C_VEL
LIN {X 0,Y 260.593,Z 728.559,A -85,B 0,C 180,E1 10399.101,E2 10399.101} C_VEL
LIN {X 0,Y 248.431,Z 741.979,A -85,B 0,C 180,E1 10396.423,E2 10396.423} C_VEL
LIN {X 0,Y 236.248,Z 754.765,A -85,B 0,C 180,E1 10392.953,E2 10392.953} C_VEL
LIN {X 0,Y 225.689,Z 765.571,A -85,B 0,C 180,E1 10388.984,E2 10388.984} C_VEL
LIN {X 0,Y 216.478,Z 775.056,A -85,B 0,C 180,E1 10384.298,E2 10384.298} C_VEL
LIN {X 0,Y 209.105,Z 783.116,A -85,B 0,C 180,E1 10378.878,E2 10378.878} C_VEL
LIN {X 0,Y 204.22,Z 789.382,A -85,B 0,C 180,E1 10373.01,E2 10373.01} C_VEL
LIN {X 0,Y 202.312,Z 793.057,A -85,B 0,C 180,E1 10368.29,E2 10368.29} C_VEL
LIN {X 0,Y 201.231,Z 802.561,A -85,B 0,C 180,E1 10363.798,E2 10363.798} C_VEL
LIN {X 0,Y 200.871,Z 810.252,A -85,B 0,C 180,E1 10359.165,E2 10359.165} C_VEL
LIN {X 0,Y 201.016,Z 815.719,A -85,B 0,C 180,E1 10354.851,E2 10354.851} C_VEL
LIN {X 0,Y 201.083,Z 819.386,A -85,B 0,C 180,E1 10350.855,E2 10350.855} C_VEL
LIN {X 0,Y 200.75,Z 821.674,A -85,B 0,C 180,E1 10346.859,E2 10346.859} C_VEL
LIN {X 0,Y 200.326,Z 823.01,A -85,B 0,C 180,E1 10341.966,E2 10341.966} C_VEL
LIN {X 0,Y 200.785,Z 822.817,A -85,B 0,C 180,E1 10336.464,E2 10336.464} C_VEL
LIN {X 0,Y 203.147,Z 820.717,A -85,B 0,C 180,E1 10330.446,E2 10330.446} C_VEL
LIN {X 0,Y 207.725,Z 816.814,A -85,B 0,C 180,E1 10324.634,E2 10324.634} C_VEL
LIN {X 0,Y 214.973,Z 810.874,A -85,B 0,C 180,E1 10318.917,E2 10318.917} C_VEL
LIN {X 0,Y 224.645,Z 803.137,A -85,B 0,C 180,E1 10313.703,E2 10313.703} C_VEL
LIN {X 0,Y 236.598,Z 793.663,A -85,B 0,C 180,E1 10309.078,E2 10309.078} C_VEL
LIN {X 0,Y 250.65,Z 782.478,A -85,B 0,C 180,E1 10305.084,E2 10305.084} C_VEL
LIN {X 0,Y 258.614,Z 776.062,A -85,B 0,C 180,E1 10303.258,E2 10303.258} C_VEL
LIN {X 0,Y 244.825,Z 785.355,A -85,B 0,C 180,E1 10299.576,E2 10299.576} C_VEL
LIN {X 0,Y 232.362,Z 793.174,A -85,B 0,C 180,E1 10295.212,E2 10295.212} C_VEL
LIN {X 0,Y 221.856,Z 799.096,A -85,B 0,C 180,E1 10290.315,E2 10290.315} C_VEL
LIN {X 0,Y 213.451,Z 803.151,A -85,B 0,C 180,E1 10284.934,E2 10284.934} C_VEL
LIN {X 0,Y 207.232,Z 805.304,A -85,B 0,C 180,E1 10279.152,E2 10279.152} C_VEL
LIN {X 0,Y 203.454,Z 805.54,A -85,B 0,C 180,E1 10273.644,E2 10273.644} C_VEL
LIN {X 0,Y 201.308,Z 804.04,A -85,B 0,C 180,E1 10267.994,E2 10267.994} C_VEL
LIN {X 0,Y 200.466,Z 801.105,A -85,B 0,C 180,E1 10262.859,E2 10262.859} C_VEL
LIN {X 0,Y 200.25,Z 796.828,A -85,B 0,C 180,E1 10257.997,E2 10257.997} C_VEL
LIN {X 0,Y 200.398,Z 790.905,A -85,B 0,C 180,E1 10253.122,E2 10253.122} C_VEL
LIN {X 0,Y 201.061,Z 783.122,A -85,B 0,C 180,E1 10248.235,E2 10248.235} C_VEL
LIN {X 0,Y 202.348,Z 773.85,A -85,B 0,C 180,E1 10243.641,E2 10243.641} C_VEL
LIN {X 0,Y 204.289,Z 763.189,A -85,B 0,C 180,E1 10239.366,E2 10239.366} C_VEL
LIN {X 0,Y 207.012,Z 750.284,A -85,B 0,C 180,E1 10235.152,E2 10235.152} C_VEL
LIN {X 0,Y 210.295,Z 735.695,A -85,B 0,C 180,E1 10231.3,E2 10231.3} C_VEL
LIN {X 0,Y 213.993,Z 719.419,A -85,B 0,C 180,E1 10227.815,E2 10227.815} C_VEL
LIN {X 0,Y 217.789,Z 701.998,A -85,B 0,C 180,E1 10224.805,E2 10224.805} C_VEL
LIN {X 0,Y 221.522,Z 683.424,A -85,B 0,C 180,E1 10222.246,E2 10222.246} C_VEL
LIN {X 0,Y 224.885,Z 664.434,A -85,B 0,C 180,E1 10220.19,E2 10220.19} C_VEL
LIN {X 0,Y 228,Z 643.45,A -85,B 0,C 180,E1 10218.449,E2 10218.449} C_VEL
LIN {X 0,Y 230.435,Z 622.363,A -85,B 0,C 180,E1 10217.194,E2 10217.194} C_VEL
LIN {X 0,Y 244.584,Z 485.544,A -85,B 0,C 180,E1 10211.122,E2 10211.122} C_VEL
LIN {X 0,Y 232.509,Z 459.851,A -85,B 0,C 180,E1 10207.597,E2 10207.597} C_VEL
LIN {X 0,Y 221.236,Z 437.773,A -85,B 0,C 180,E1 10204.006,E2 10204.006} C_VEL
LIN {X 0,Y 211.636,Z 420.411,A -85,B 0,C 180,E1 10200.68,E2 10200.68} C_VEL
LIN {X 0,Y 206.141,Z 408.815,A -85,B 0,C 180,E1 10197.125,E2 10197.125} C_VEL
LIN {X 0,Y 204.193,Z 404.853,A -85,B 0,C 180,E1 10195.836,E2 10195.836} C_VEL
LIN {X 0,Y 202.98,Z 401.512,A -85,B 0,C 180,E1 10194.753,E2 10194.753} C_VEL
LIN {X 0,Y 202.978,Z 401.514,A -85,B 0,C 180,E1 10189.57,E2 10189.57} C_VEL
LIN {X 0,Y 202.992,Z 401.508,A -85,B 0,C 180,E1 10183.967,E2 10183.967} C_VEL
LIN {X 0,Y 202.991,Z 401.504,A -85,B 0,C 180,E1 10178.086,E2 10178.086} C_VEL
LIN {X 0,Y 202.979,Z 401.508,A -85,B 0,C 180,E1 10172.258,E2 10172.258} C_VEL
LIN {X 0,Y 202.967,Z 401.505,A -85,B 0,C 180,E1 10166.894,E2 10166.894} C_VEL
LIN {X 0,Y 202.979,Z 401.505,A -85,B 0,C 180,E1 10161.502,E2 10161.502} C_VEL
LIN {X 0,Y 202.996,Z 401.513,A -85,B 0,C 180,E1 10155.743,E2 10155.743} C_VEL
LIN {X 0,Y 202.98,Z 401.514,A -85,B 0,C 180,E1 10150.13,E2 10150.13} C_VEL
LIN {X 0,Y 202.972,Z 401.514,A -85,B 0,C 180,E1 10144.935,E2 10144.935} C_VEL
LIN {X 0,Y 202.993,Z 401.551,A -85,B 0,C 180,E1 10139.37,E2 10139.37} C_VEL
LIN {X 0,Y 206.9,Z 413.747,A -85,B 0,C 180,E1 10134.215,E2 10134.215} C_VEL
LIN {X 0,Y 210.689,Z 426.254,A -85,B 0,C 180,E1 10129.404,E2 10129.404} C_VEL
LIN {X 0,Y 214.586,Z 440.736,A -85,B 0,C 180,E1 10124.341,E2 10124.341} C_VEL
LIN {X 0,Y 218.228,Z 455.976,A -85,B 0,C 180,E1 10119.464,E2 10119.464} C_VEL
LIN {X 0,Y 219.154,Z 461.298,A -85,B 0,C 180,E1 10117.881,E2 10117.881} C_VEL
LIN {X 0,Y 215.805,Z 475.91,A -85,B 0,C 180,E1 10114.35,E2 10114.35} C_VEL
LIN {X 0,Y 217.515,Z 509.095,A -85,B 0,C 180,E1 10112.133,E2 10112.133} C_VEL
LIN {X 0,Y 218.475,Z 523.982,A -85,B 0,C 180,E1 10111.142,E2 10111.142} C_VEL
LIN {X 0,Y 211.484,Z 617.152,A -85,B 0,C 180,E1 10105.854,E2 10105.854} C_VEL
LIN {X 0,Y 210.05,Z 636.495,A -85,B 0,C 180,E1 10104.24,E2 10104.24} C_VEL
LIN {X 0,Y 208.418,Z 653.993,A -85,B 0,C 180,E1 10102.272,E2 10102.272} C_VEL
LIN {X 0,Y 206.707,Z 670.96,A -85,B 0,C 180,E1 10099.792,E2 10099.792} C_VEL
LIN {X 0,Y 205.03,Z 687.371,A -85,B 0,C 180,E1 10096.722,E2 10096.722} C_VEL
LIN {X 0,Y 203.631,Z 702.215,A -85,B 0,C 180,E1 10093.227,E2 10093.227} C_VEL
LIN {X 0,Y 202.694,Z 715.285,A -85,B 0,C 180,E1 10089.369,E2 10089.369} C_VEL
LIN {X 0,Y 202.335,Z 725.218,A -85,B 0,C 180,E1 10085.672,E2 10085.672} C_VEL
LIN {X 0,Y 202.521,Z 733.881,A -85,B 0,C 180,E1 10081.698,E2 10081.698} C_VEL
LIN {X 0,Y 203.416,Z 740.966,A -85,B 0,C 180,E1 10077.465,E2 10077.465} C_VEL
LIN {X 0,Y 205.309,Z 746.541,A -85,B 0,C 180,E1 10073.007,E2 10073.007} C_VEL
LIN {X 0,Y 208.113,Z 749.95,A -85,B 0,C 180,E1 10068.85,E2 10068.85} C_VEL
LIN {X 0,Y 208.963,Z 751.22,A -85,B 0,C 180,E1 10066.756,E2 10066.756} C_VEL
LIN {X 0,Y 209.06,Z 753.529,A -85,B 0,C 180,E1 10061.432,E2 10061.432} C_VEL
LIN {X 0,Y 210.878,Z 753.721,A -85,B 0,C 180,E1 10059.381,E2 10059.381} C_VEL
LIN {X 0,Y 211.09,Z 753.713,A -85,B 0,C 180,E1 10059.242,E2 10059.242} C_VEL
LIN {X 0,Y 218.448,Z 752.141,A -85,B 0,C 180,E1 10055.097,E2 10055.097} C_VEL
LIN {X 0,Y 226.976,Z 748.795,A -85,B 0,C 180,E1 10051.304,E2 10051.304} C_VEL
LIN {X 0,Y 236.667,Z 743.661,A -85,B 0,C 180,E1 10047.838,E2 10047.838} C_VEL
LIN {X 0,Y 248.098,Z 736.207,A -85,B 0,C 180,E1 10044.526,E2 10044.526} C_VEL
LIN {X 0,Y 259.31,Z 727.659,A -85,B 0,C 180,E1 10041.869,E2 10041.869} C_VEL
LIN {X 0,Y 261.396,Z 725.968,A -85,B 0,C 180,E1 10041.386,E2 10041.386} C_VEL
LIN {X 0,Y 248.936,Z 738.679,A -85,B 0,C 180,E1 10039.035,E2 10039.035} C_VEL
LIN {X 0,Y 236.345,Z 750.791,A -85,B 0,C 180,E1 10035.988,E2 10035.988} C_VEL
LIN {X 0,Y 224.536,Z 761.693,A -85,B 0,C 180,E1 10032.253,E2 10032.253} C_VEL
LIN {X 0,Y 213.937,Z 771.351,A -85,B 0,C 180,E1 10027.752,E2 10027.752} C_VEL
LIN {X 0,Y 205.035,Z 779.668,A -85,B 0,C 180,E1 10022.44,E2 10022.44} C_VEL
LIN {X 0,Y 198.643,Z 786.163,A -85,B 0,C 180,E1 10016.614,E2 10016.614} C_VEL
LIN {X 0,Y 194.923,Z 790.921,A -85,B 0,C 180,E1 10010.415,E2 10010.415} C_VEL
LIN {X 0,Y 194.347,Z 792.283,A -85,B 0,C 180,E1 10008.29,E2 10008.29} C_VEL
LIN {X 0,Y 193.254,Z 802.079,A -85,B 0,C 180,E1 10003.463,E2 10003.463} C_VEL
LIN {X 0,Y 192.959,Z 809.726,A -85,B 0,C 180,E1 9998.643,E2 9998.643} C_VEL
LIN {X 0,Y 193.134,Z 815.14,A -85,B 0,C 180,E1 9994.156,E2 9994.156} C_VEL
LIN {X 0,Y 193.154,Z 818.738,A -85,B 0,C 180,E1 9990,E2 9990} C_VEL
LIN {X 0,Y 192.677,Z 821.086,A -85,B 0,C 180,E1 9985.536,E2 9985.536} C_VEL
LIN {X 0,Y 192.366,Z 822.33,A -85,B 0,C 180,E1 9980.124,E2 9980.124} C_VEL
LIN {X 0,Y 193.464,Z 821.911,A -85,B 0,C 180,E1 9974.004,E2 9974.004} C_VEL
LIN {X 0,Y 196.668,Z 819.697,A -85,B 0,C 180,E1 9967.9,E2 9967.9} C_VEL
LIN {X 0,Y 202.613,Z 815.515,A -85,B 0,C 180,E1 9961.722,E2 9961.722} C_VEL
LIN {X 0,Y 211.128,Z 809.558,A -85,B 0,C 180,E1 9956.025,E2 9956.025} C_VEL
LIN {X 0,Y 222.07,Z 801.921,A -85,B 0,C 180,E1 9950.924,E2 9950.924} C_VEL
LIN {X 0,Y 235.243,Z 792.668,A -85,B 0,C 180,E1 9946.484,E2 9946.484} C_VEL
LIN {X 0,Y 248.299,Z 783.385,A -85,B 0,C 180,E1 9943.13,E2 9943.13} C_VEL
LIN {X 0,Y 234.268,Z 791.459,A -85,B 0,C 180,E1 9939.173,E2 9939.173} C_VEL
LIN {X 0,Y 221.452,Z 798.126,A -85,B 0,C 180,E1 9934.359,E2 9934.359} C_VEL
LIN {X 0,Y 210.89,Z 802.893,A -85,B 0,C 180,E1 9928.92,E2 9928.92} C_VEL
LIN {X 0,Y 203.039,Z 805.604,A -85,B 0,C 180,E1 9923.201,E2 9923.201} C_VEL
LIN {X 0,Y 197.672,Z 806.427,A -85,B 0,C 180,E1 9917.363,E2 9917.363} C_VEL
LIN {X 0,Y 194.323,Z 805.405,A -85,B 0,C 180,E1 9911.275,E2 9911.275} C_VEL
LIN {X 0,Y 192.806,Z 802.825,A -85,B 0,C 180,E1 9905.654,E2 9905.654} C_VEL
LIN {X 0,Y 192.316,Z 798.793,A -85,B 0,C 180,E1 9900.298,E2 9900.298} C_VEL
LIN {X 0,Y 192.289,Z 793.369,A -85,B 0,C 180,E1 9895.227,E2 9895.227} C_VEL
LIN {X 0,Y 192.724,Z 786.163,A -85,B 0,C 180,E1 9890.142,E2 9890.142} C_VEL
LIN {X 0,Y 193.757,Z 777.502,A -85,B 0,C 180,E1 9885.353,E2 9885.353} C_VEL
LIN {X 0,Y 195.587,Z 766.758,A -85,B 0,C 180,E1 9880.592,E2 9880.592} C_VEL
LIN {X 0,Y 198.123,Z 754.468,A -85,B 0,C 180,E1 9876.188,E2 9876.188} C_VEL
LIN {X 0,Y 201.384,Z 740.156,A -85,B 0,C 180,E1 9872.018,E2 9872.018} C_VEL
LIN {X 0,Y 204.989,Z 724.748,A -85,B 0,C 180,E1 9868.375,E2 9868.375} C_VEL
LIN {X 0,Y 208.72,Z 708.395,A -85,B 0,C 180,E1 9865.245,E2 9865.245} C_VEL
LIN {X 0,Y 212.569,Z 690.359,A -85,B 0,C 180,E1 9862.473,E2 9862.473} C_VEL
LIN {X 0,Y 216.407,Z 670.348,A -85,B 0,C 180,E1 9860.042,E2 9860.042} C_VEL
LIN {X 0,Y 219.659,Z 650.328,A -85,B 0,C 180,E1 9858.175,E2 9858.175} C_VEL
LIN {X 0,Y 222.413,Z 629,A -85,B 0,C 180,E1 9856.727,E2 9856.727} C_VEL
LIN {X 0,Y 237.61,Z 487.944,A -85,B 0,C 180,E1 9850.19,E2 9850.19} C_VEL
LIN {X 0,Y 225.845,Z 462.682,A -85,B 0,C 180,E1 9846.585,E2 9846.585} C_VEL
LIN {X 0,Y 214.484,Z 440.464,A -85,B 0,C 180,E1 9842.815,E2 9842.815} C_VEL
LIN {X 0,Y 204.038,Z 421.721,A -85,B 0,C 180,E1 9839.022,E2 9839.022} C_VEL
LIN {X 0,Y 198.464,Z 410.176,A -85,B 0,C 180,E1 9835.355,E2 9835.355} C_VEL
LIN {X 0,Y 196.548,Z 406.257,A -85,B 0,C 180,E1 9834.015,E2 9834.015} C_VEL
LIN {X 0,Y 195.064,Z 402.695,A -85,B 0,C 180,E1 9832.84,E2 9832.84} C_VEL
LIN {X 0,Y 195.034,Z 402.497,A -85,B 0,C 180,E1 9827.298,E2 9827.298} C_VEL
LIN {X 0,Y 195.041,Z 402.502,A -85,B 0,C 180,E1 9821.72,E2 9821.72} C_VEL
LIN {X 0,Y 195.048,Z 402.501,A -85,B 0,C 180,E1 9815.885,E2 9815.885} C_VEL
LIN {X 0,Y 195.056,Z 402.497,A -85,B 0,C 180,E1 9810,E2 9810} C_VEL
LIN {X 0,Y 195.047,Z 402.499,A -85,B 0,C 180,E1 9803.988,E2 9803.988} C_VEL
LIN {X 0,Y 195.04,Z 402.498,A -85,B 0,C 180,E1 9798.167,E2 9798.167} C_VEL
LIN {X 0,Y 195.032,Z 402.5,A -85,B 0,C 180,E1 9792.702,E2 9792.702} C_VEL
LIN {X 0,Y 195.036,Z 402.504,A -85,B 0,C 180,E1 9787.069,E2 9787.069} C_VEL
LIN {X 0,Y 195.051,Z 402.504,A -85,B 0,C 180,E1 9781.528,E2 9781.528} C_VEL
LIN {X 0,Y 195.043,Z 402.551,A -85,B 0,C 180,E1 9781.024,E2 9781.024} C_VEL
LIN {X 0,Y 198.691,Z 413.652,A -85,B 0,C 180,E1 9776.042,E2 9776.042} C_VEL
LIN {X 0,Y 202.366,Z 425.714,A -85,B 0,C 180,E1 9771.135,E2 9771.135} C_VEL
LIN {X 0,Y 205.921,Z 438.655,A -85,B 0,C 180,E1 9766.343,E2 9766.343} C_VEL
LIN {X 0,Y 209.576,Z 453.583,A -85,B 0,C 180,E1 9761.287,E2 9761.287} C_VEL
LIN {X 0,Y 211.498,Z 462.621,A -85,B 0,C 180,E1 9758.439,E2 9758.439} C_VEL
LIN {X 0,Y 208.338,Z 475.935,A -85,B 0,C 180,E1 9755.152,E2 9755.152} C_VEL
LIN {X 0,Y 209.808,Z 508.149,A -85,B 0,C 180,E1 9752.916,E2 9752.916} C_VEL
LIN {X 0,Y 210.837,Z 524.398,A -85,B 0,C 180,E1 9751.785,E2 9751.785} C_VEL
LIN {X 0,Y 203.593,Z 618.183,A -85,B 0,C 180,E1 9746.242,E2 9746.242} C_VEL
LIN {X 0,Y 202.105,Z 637.335,A -85,B 0,C 180,E1 9744.555,E2 9744.555} C_VEL
LIN {X 0,Y 200.339,Z 655.56,A -85,B 0,C 180,E1 9742.384,E2 9742.384} C_VEL
LIN {X 0,Y 198.562,Z 672.812,A -85,B 0,C 180,E1 9739.718,E2 9739.718} C_VEL
LIN {X 0,Y 196.943,Z 688.451,A -85,B 0,C 180,E1 9736.67,E2 9736.67} C_VEL
LIN {X 0,Y 195.58,Z 702.866,A -85,B 0,C 180,E1 9733.15,E2 9733.15} C_VEL
LIN {X 0,Y 194.705,Z 714.953,A -85,B 0,C 180,E1 9729.459,E2 9729.459} C_VEL
LIN {X 0,Y 194.335,Z 725.303,A -85,B 0,C 180,E1 9725.61,E2 9725.61} C_VEL
LIN {X 0,Y 194.544,Z 734.145,A -85,B 0,C 180,E1 9721.473,E2 9721.473} C_VEL
LIN {X 0,Y 195.514,Z 741.592,A -85,B 0,C 180,E1 9717.069,E2 9717.069} C_VEL
LIN {X 0,Y 197.547,Z 747.396,A -85,B 0,C 180,E1 9712.439,E2 9712.439} C_VEL
LIN {X 0,Y 200.743,Z 751.307,A -85,B 0,C 180,E1 9707.925,E2 9707.925} C_VEL
LIN {X 0,Y 205.473,Z 753.431,A -85,B 0,C 180,E1 9703.316,E2 9703.316} C_VEL
LIN {X 0,Y 211.09,Z 753.713,A -85,B 0,C 180,E1 9699.242,E2 9699.242} C_VEL
LIN {X 0,Y 213.535,Z 753.694,A -85,B 0,C 180,E1 9697.091,E2 9697.091} C_VEL
LIN {X 0,Y 217.071,Z 753.182,A -85,B 0,C 180,E1 9692.431,E2 9692.431} C_VEL
LIN {X 0,Y 219.986,Z 752.071,A -85,B 0,C 180,E1 9690.577,E2 9690.577} C_VEL
LIN {X 0,Y 220.836,Z 751.719,A -85,B 0,C 180,E1 9690.219,E2 9690.219} C_VEL
LIN {X 0,Y 231.775,Z 746.742,A -85,B 0,C 180,E1 9686.483,E2 9686.483} C_VEL
LIN {X 0,Y 243.065,Z 740.319,A -85,B 0,C 180,E1 9683.383,E2 9683.383} C_VEL
LIN {X 0,Y 250.417,Z 735.526,A -85,B 0,C 180,E1 9681.628,E2 9681.628} C_VEL
LIN {X 0,Y 236.595,Z 747.759,A -85,B 0,C 180,E1 9678.785,E2 9678.785} C_VEL
LIN {X 0,Y 223.048,Z 759.127,A -85,B 0,C 180,E1 9675.095,E2 9675.095} C_VEL
LIN {X 0,Y 211.275,Z 768.677,A -85,B 0,C 180,E1 9670.775,E2 9670.775} C_VEL
LIN {X 0,Y 201.066,Z 776.973,A -85,B 0,C 180,E1 9665.579,E2 9665.579} C_VEL
LIN {X 0,Y 193.028,Z 783.795,A -85,B 0,C 180,E1 9659.478,E2 9659.478} C_VEL
LIN {X 0,Y 188.131,Z 788.617,A -85,B 0,C 180,E1 9653.156,E2 9653.156} C_VEL
LIN {X 0,Y 186.441,Z 791.096,A -85,B 0,C 180,E1 9648.446,E2 9648.446} C_VEL
LIN {X 0,Y 185.372,Z 800.447,A -85,B 0,C 180,E1 9643.729,E2 9643.729} C_VEL
LIN {X 0,Y 185.052,Z 808.311,A -85,B 0,C 180,E1 9638.702,E2 9638.702} C_VEL
LIN {X 0,Y 185.239,Z 813.919,A -85,B 0,C 180,E1 9634.024,E2 9634.024} C_VEL
LIN {X 0,Y 185.27,Z 817.367,A -85,B 0,C 180,E1 9630,E2 9630} C_VEL
LIN {X 0,Y 184.737,Z 820,A -85,B 0,C 180,E1 9625.343,E2 9625.343} C_VEL
LIN {X 0,Y 184.43,Z 821.499,A -85,B 0,C 180,E1 9619.694,E2 9619.694} C_VEL
LIN {X 0,Y 185.749,Z 821.38,A -85,B 0,C 180,E1 9613.102,E2 9613.102} C_VEL
LIN {X 0,Y 189.628,Z 819.326,A -85,B 0,C 180,E1 9606.376,E2 9606.376} C_VEL
LIN {X 0,Y 196.616,Z 815.247,A -85,B 0,C 180,E1 9599.771,E2 9599.771} C_VEL
LIN {X 0,Y 206.469,Z 809.329,A -85,B 0,C 180,E1 9593.786,E2 9593.786} C_VEL
LIN {X 0,Y 218.964,Z 801.685,A -85,B 0,C 180,E1 9588.538,E2 9588.538} C_VEL
LIN {X 0,Y 233.817,Z 792.394,A -85,B 0,C 180,E1 9584.076,E2 9584.076} C_VEL
LIN {X 0,Y 237.93,Z 789.744,A -85,B 0,C 180,E1 9583.027,E2 9583.027} C_VEL
LIN {X 0,Y 223.638,Z 796.69,A -85,B 0,C 180,E1 9578.75,E2 9578.75} C_VEL
LIN {X 0,Y 211.036,Z 802.063,A -85,B 0,C 180,E1 9573.664,E2 9573.664} C_VEL
LIN {X 0,Y 200.78,Z 805.58,A -85,B 0,C 180,E1 9567.911,E2 9567.911} C_VEL
LIN {X 0,Y 193.323,Z 807.085,A -85,B 0,C 180,E1 9561.862,E2 9561.862} C_VEL
LIN {X 0,Y 188.436,Z 806.769,A -85,B 0,C 180,E1 9555.7,E2 9555.7} C_VEL
LIN {X 0,Y 185.702,Z 804.779,A -85,B 0,C 180,E1 9549.608,E2 9549.608} C_VEL
LIN {X 0,Y 184.547,Z 801.241,A -85,B 0,C 180,E1 9543.727,E2 9543.727} C_VEL
LIN {X 0,Y 184.269,Z 796.568,A -85,B 0,C 180,E1 9538.445,E2 9538.445} C_VEL
LIN {X 0,Y 184.391,Z 790.648,A -85,B 0,C 180,E1 9533.461,E2 9533.461} C_VEL
LIN {X 0,Y 185.013,Z 783.039,A -85,B 0,C 180,E1 9528.465,E2 9528.465} C_VEL
LIN {X 0,Y 186.342,Z 773.531,A -85,B 0,C 180,E1 9523.478,E2 9523.478} C_VEL
LIN {X 0,Y 188.399,Z 762.581,A -85,B 0,C 180,E1 9518.845,E2 9518.845} C_VEL
LIN {X 0,Y 191.318,Z 749.321,A -85,B 0,C 180,E1 9514.292,E2 9514.292} C_VEL
LIN {X 0,Y 194.873,Z 734.324,A -85,B 0,C 180,E1 9510.125,E2 9510.125} C_VEL
LIN {X 0,Y 198.832,Z 717.784,A -85,B 0,C 180,E1 9506.416,E2 9506.416} C_VEL
LIN {X 0,Y 202.909,Z 699.932,A -85,B 0,C 180,E1 9503.222,E2 9503.222} C_VEL
LIN {X 0,Y 206.877,Z 681.032,A -85,B 0,C 180,E1 9500.538,E2 9500.538} C_VEL
LIN {X 0,Y 210.546,Z 661.079,A -85,B 0,C 180,E1 9498.329,E2 9498.329} C_VEL
LIN {X 0,Y 213.657,Z 640.518,A -85,B 0,C 180,E1 9496.616,E2 9496.616} C_VEL
LIN {X 0,Y 216.441,Z 616.721,A -85,B 0,C 180,E1 9495.212,E2 9495.212} C_VEL
LIN {X 0,Y 230.661,Z 490.328,A -85,B 0,C 180,E1 9489.223,E2 9489.223} C_VEL
LIN {X 0,Y 219.132,Z 465.481,A -85,B 0,C 180,E1 9485.534,E2 9485.534} C_VEL
LIN {X 0,Y 207.827,Z 443.261,A -85,B 0,C 180,E1 9481.588,E2 9481.588} C_VEL
LIN {X 0,Y 197.234,Z 424.225,A -85,B 0,C 180,E1 9477.526,E2 9477.526} C_VEL
LIN {X 0,Y 195.441,Z 421.139,A -85,B 0,C 180,E1 9476.757,E2 9476.757} C_VEL
LIN {X 0,Y 190.825,Z 411.564,A -85,B 0,C 180,E1 9473.467,E2 9473.467} C_VEL
LIN {X 0,Y 188.952,Z 407.675,A -85,B 0,C 180,E1 9472.068,E2 9472.068} C_VEL
LIN {X 0,Y 187.246,Z 404.31,A -85,B 0,C 180,E1 9470.8,E2 9470.8} C_VEL
LIN {X 0,Y 187.106,Z 403.485,A -85,B 0,C 180,E1 9470.453,E2 9470.453} C_VEL
LIN {X 0,Y 187.103,Z 403.492,A -85,B 0,C 180,E1 9464.546,E2 9464.546} C_VEL
LIN {X 0,Y 187.092,Z 403.483,A -85,B 0,C 180,E1 9458.916,E2 9458.916} C_VEL
LIN {X 0,Y 187.092,Z 403.48,A -85,B 0,C 180,E1 9453.37,E2 9453.37} C_VEL
LIN {X 0,Y 187.103,Z 403.476,A -85,B 0,C 180,E1 9447.856,E2 9447.856} C_VEL
LIN {X 0,Y 187.11,Z 403.479,A -85,B 0,C 180,E1 9442.014,E2 9442.014} C_VEL
LIN {X 0,Y 187.107,Z 403.49,A -85,B 0,C 180,E1 9436.086,E2 9436.086} C_VEL
LIN {X 0,Y 187.102,Z 403.491,A -85,B 0,C 180,E1 9430.142,E2 9430.142} C_VEL
LIN {X 0,Y 187.094,Z 403.493,A -85,B 0,C 180,E1 9424.578,E2 9424.578} C_VEL
LIN {X 0,Y 187.116,Z 403.656,A -85,B 0,C 180,E1 9422.753,E2 9422.753} C_VEL
LIN {X 0,Y 190.793,Z 414.638,A -85,B 0,C 180,E1 9417.537,E2 9417.537} C_VEL
LIN {X 0,Y 194.553,Z 426.895,A -85,B 0,C 180,E1 9412.296,E2 9412.296} C_VEL
LIN {X 0,Y 198.241,Z 440.405,A -85,B 0,C 180,E1 9407.086,E2 9407.086} C_VEL
LIN {X 0,Y 201.649,Z 454.397,A -85,B 0,C 180,E1 9402.158,E2 9402.158} C_VEL
LIN {X 0,Y 203.734,Z 464.304,A -85,B 0,C 180,E1 9398.917,E2 9398.917} C_VEL
LIN {X 0,Y 200.892,Z 475.766,A -85,B 0,C 180,E1 9396.01,E2 9396.01} C_VEL
LIN {X 0,Y 202.135,Z 507.053,A -85,B 0,C 180,E1 9393.767,E2 9393.767} C_VEL
LIN {X 0,Y 203.201,Z 525.002,A -85,B 0,C 180,E1 9392.458,E2 9392.458} C_VEL
LIN {X 0,Y 195.749,Z 618.017,A -85,B 0,C 180,E1 9386.689,E2 9386.689} C_VEL
LIN {X 0,Y 194.175,Z 637.766,A -85,B 0,C 180,E1 9384.895,E2 9384.895} C_VEL
LIN {X 0,Y 192.348,Z 656.192,A -85,B 0,C 180,E1 9382.623,E2 9382.623} C_VEL
LIN {X 0,Y 190.504,Z 673.789,A -85,B 0,C 180,E1 9379.801,E2 9379.801} C_VEL
LIN {X 0,Y 188.855,Z 689.409,A -85,B 0,C 180,E1 9376.608,E2 9376.608} C_VEL
LIN {X 0,Y 187.452,Z 704.298,A -85,B 0,C 180,E1 9372.789,E2 9372.789} C_VEL
LIN {X 0,Y 186.578,Z 717.284,A -85,B 0,C 180,E1 9368.63,E2 9368.63} C_VEL
LIN {X 0,Y 186.331,Z 727.328,A -85,B 0,C 180,E1 9364.617,E2 9364.617} C_VEL
LIN {X 0,Y 186.768,Z 736.651,A -85,B 0,C 180,E1 9360,E2 9360} C_VEL
LIN {X 0,Y 188.06,Z 743.783,A -85,B 0,C 180,E1 9355.426,E2 9355.426} C_VEL
LIN {X 0,Y 190.545,Z 749.458,A -85,B 0,C 180,E1 9350.639,E2 9350.639} C_VEL
LIN {X 0,Y 194.291,Z 753.192,A -85,B 0,C 180,E1 9346.003,E2 9346.003} C_VEL
LIN {X 0,Y 199.667,Z 755.268,A -85,B 0,C 180,E1 9341.308,E2 9341.308} C_VEL
LIN {X 0,Y 206.446,Z 755.457,A -85,B 0,C 180,E1 9336.903,E2 9336.903} C_VEL
LIN {X 0,Y 215.053,Z 753.683,A -85,B 0,C 180,E1 9332.595,E2 9332.595} C_VEL
LIN {X 0,Y 220.836,Z 751.719,A -85,B 0,C 180,E1 9330.219,E2 9330.219} C_VEL
LIN {X 0,Y 224.9,Z 750.132,A -85,B 0,C 180,E1 9328.227,E2 9328.227} C_VEL
LIN {X 0,Y 232.132,Z 747.345,A -85,B 0,C 180,E1 9324.043,E2 9324.043} C_VEL
LIN {X 0,Y 236.104,Z 745.404,A -85,B 0,C 180,E1 9322.67,E2 9322.67} C_VEL
LIN {X 0,Y 236.817,Z 745.009,A -85,B 0,C 180,E1 9322.49,E2 9322.49} C_VEL
LIN {X 0,Y 239.341,Z 743.684,A -85,B 0,C 180,E1 9321.853,E2 9321.853} C_VEL
LIN {X 0,Y 225.042,Z 754.703,A -85,B 0,C 180,E1 9318.666,E2 9318.666} C_VEL
LIN {X 0,Y 211.773,Z 764.417,A -85,B 0,C 180,E1 9314.708,E2 9314.708} C_VEL
LIN {X 0,Y 199.845,Z 772.917,A -85,B 0,C 180,E1 9309.822,E2 9309.822} C_VEL
LIN {X 0,Y 190.254,Z 779.792,A -85,B 0,C 180,E1 9304.217,E2 9304.217} C_VEL
LIN {X 0,Y 183.053,Z 785.302,A -85,B 0,C 180,E1 9297.664,E2 9297.664} C_VEL
LIN {X 0,Y 179.028,Z 789.072,A -85,B 0,C 180,E1 9290.601,E2 9290.601} C_VEL
LIN {X 0,Y 178.552,Z 789.83,A -85,B 0,C 180,E1 9288.614,E2 9288.614} C_VEL
LIN {X 0,Y 177.415,Z 799.827,A -85,B 0,C 180,E1 9283.36,E2 9283.36} C_VEL
LIN {X 0,Y 177.159,Z 807.255,A -85,B 0,C 180,E1 9278.438,E2 9278.438} C_VEL
LIN {X 0,Y 177.37,Z 812.611,A -85,B 0,C 180,E1 9273.83,E2 9273.83} C_VEL
LIN {X 0,Y 177.374,Z 816.184,A -85,B 0,C 180,E1 9269.677,E2 9269.677} C_VEL
LIN {X 0,Y 176.822,Z 818.765,A -85,B 0,C 180,E1 9265.134,E2 9265.134} C_VEL
LIN {X 0,Y 176.535,Z 820.577,A -85,B 0,C 180,E1 9258.897,E2 9258.897} C_VEL
LIN {X 0,Y 178.132,Z 820.716,A -85,B 0,C 180,E1 9252.018,E2 9252.018} C_VEL
LIN {X 0,Y 182.475,Z 818.995,A -85,B 0,C 180,E1 9245.044,E2 9245.044} C_VEL
LIN {X 0,Y 190.073,Z 815.338,A -85,B 0,C 180,E1 9238.262,E2 9238.262} C_VEL
LIN {X 0,Y 200.598,Z 809.939,A -85,B 0,C 180,E1 9232.187,E2 9232.187} C_VEL
LIN {X 0,Y 213.771,Z 802.908,A -85,B 0,C 180,E1 9226.931,E2 9226.931} C_VEL
LIN {X 0,Y 227.524,Z 795.324,A -85,B 0,C 180,E1 9222.933,E2 9222.933} C_VEL
LIN {X 0,Y 212.963,Z 801.176,A -85,B 0,C 180,E1 9218.297,E2 9218.297} C_VEL
LIN {X 0,Y 200.596,Z 805.267,A -85,B 0,C 180,E1 9212.908,E2 9212.908} C_VEL
LIN {X 0,Y 190.675,Z 807.499,A -85,B 0,C 180,E1 9206.805,E2 9206.805} C_VEL
LIN {X 0,Y 183.68,Z 807.855,A -85,B 0,C 180,E1 9200.388,E2 9200.388} C_VEL
LIN {X 0,Y 179.173,Z 806.33,A -85,B 0,C 180,E1 9193.555,E2 9193.555} C_VEL
LIN {X 0,Y 177.056,Z 803.192,A -85,B 0,C 180,E1 9187.136,E2 9187.136} C_VEL
LIN {X 0,Y 176.383,Z 798.777,A -85,B 0,C 180,E1 9181.299,E2 9181.299} C_VEL
LIN {X 0,Y 176.304,Z 793.012,A -85,B 0,C 180,E1 9175.772,E2 9175.772} C_VEL
LIN {X 0,Y 176.691,Z 785.946,A -85,B 0,C 180,E1 9170.554,E2 9170.554} C_VEL
LIN {X 0,Y 177.737,Z 777.036,A -85,B 0,C 180,E1 9165.336,E2 9165.336} C_VEL
LIN {X 0,Y 179.682,Z 765.937,A -85,B 0,C 180,E1 9160.122,E2 9160.122} C_VEL
LIN {X 0,Y 182.381,Z 753.445,A -85,B 0,C 180,E1 9155.376,E2 9155.376} C_VEL
LIN {X 0,Y 185.761,Z 739.343,A -85,B 0,C 180,E1 9151.025,E2 9151.025} C_VEL
LIN {X 0,Y 189.63,Z 723.58,A -85,B 0,C 180,E1 9147.105,E2 9147.105} C_VEL
LIN {X 0,Y 193.822,Z 706.078,A -85,B 0,C 180,E1 9143.612,E2 9143.612} C_VEL
LIN {X 0,Y 197.969,Z 687.545,A -85,B 0,C 180,E1 9140.664,E2 9140.664} C_VEL
LIN {X 0,Y 201.876,Z 667.932,A -85,B 0,C 180,E1 9138.228,E2 9138.228} C_VEL
LIN {X 0,Y 205.363,Z 647.091,A -85,B 0,C 180,E1 9136.261,E2 9136.261} C_VEL
LIN {X 0,Y 208.228,Z 625.545,A -85,B 0,C 180,E1 9134.772,E2 9134.772} C_VEL
LIN {X 0,Y 223.685,Z 492.52,A -85,B 0,C 180,E1 9128.192,E2 9128.192} C_VEL
LIN {X 0,Y 212.185,Z 467.788,A -85,B 0,C 180,E1 9124.353,E2 9124.353} C_VEL
LIN {X 0,Y 201.543,Z 446.748,A -85,B 0,C 180,E1 9120.441,E2 9120.441} C_VEL
LIN {X 0,Y 191.661,Z 428.92,A -85,B 0,C 180,E1 9116.49,E2 9116.49} C_VEL
LIN {X 0,Y 187.447,Z 421.543,A -85,B 0,C 180,E1 9114.586,E2 9114.586} C_VEL
LIN {X 0,Y 182.782,Z 412.354,A -85,B 0,C 180,E1 9111.164,E2 9111.164} C_VEL
LIN {X 0,Y 180.928,Z 408.577,A -85,B 0,C 180,E1 9109.701,E2 9109.701} C_VEL
LIN {X 0,Y 179.295,Z 405.215,A -85,B 0,C 180,E1 9108.366,E2 9108.366} C_VEL
LIN {X 0,Y 179.168,Z 404.477,A -85,B 0,C 180,E1 9108.096,E2 9108.096} C_VEL
LIN {X 0,Y 179.164,Z 404.475,A -85,B 0,C 180,E1 9102.243,E2 9102.243} C_VEL
LIN {X 0,Y 179.172,Z 404.48,A -85,B 0,C 180,E1 9096.086,E2 9096.086} C_VEL
LIN {X 0,Y 179.177,Z 404.475,A -85,B 0,C 180,E1 9090,E2 9090} C_VEL
LIN {X 0,Y 179.169,Z 404.476,A -85,B 0,C 180,E1 9083.913,E2 9083.913} C_VEL
LIN {X 0,Y 179.163,Z 404.473,A -85,B 0,C 180,E1 9077.756,E2 9077.756} C_VEL
LIN {X 0,Y 179.165,Z 404.482,A -85,B 0,C 180,E1 9071.789,E2 9071.789} C_VEL
LIN {X 0,Y 179.163,Z 404.476,A -85,B 0,C 180,E1 9065.959,E2 9065.959} C_VEL
LIN {X 0,Y 179.177,Z 404.641,A -85,B 0,C 180,E1 9064.691,E2 9064.691} C_VEL
LIN {X 0,Y 182.455,Z 414.428,A -85,B 0,C 180,E1 9059.724,E2 9059.724} C_VEL
LIN {X 0,Y 186.053,Z 425.762,A -85,B 0,C 180,E1 9054.521,E2 9054.521} C_VEL
LIN {X 0,Y 189.5,Z 438.051,A -85,B 0,C 180,E1 9049.446,E2 9049.446} C_VEL
LIN {X 0,Y 192.903,Z 451.656,A -85,B 0,C 180,E1 9044.333,E2 9044.333} C_VEL
LIN {X 0,Y 196.014,Z 465.565,A -85,B 0,C 180,E1 9039.53,E2 9039.53} C_VEL
LIN {X 0,Y 193.444,Z 475.724,A -85,B 0,C 180,E1 9036.886,E2 9036.886} C_VEL
LIN {X 0,Y 194.482,Z 506.578,A -85,B 0,C 180,E1 9034.58,E2 9034.58} C_VEL
LIN {X 0,Y 195.551,Z 525.543,A -85,B 0,C 180,E1 9033.147,E2 9033.147} C_VEL
LIN {X 0,Y 187.841,Z 618.882,A -85,B 0,C 180,E1 9027.088,E2 9027.088} C_VEL
LIN {X 0,Y 186.253,Z 638.198,A -85,B 0,C 180,E1 9025.264,E2 9025.264} C_VEL
LIN {X 0,Y 184.433,Z 656.078,A -85,B 0,C 180,E1 9022.976,E2 9022.976} C_VEL
LIN {X 0,Y 182.529,Z 673.78,A -85,B 0,C 180,E1 9020.021,E2 9020.021} C_VEL
LIN {X 0,Y 180.808,Z 689.833,A -85,B 0,C 180,E1 9016.626,E2 9016.626} C_VEL
LIN {X 0,Y 179.369,Z 705.177,A -85,B 0,C 180,E1 9012.557,E2 9012.557} C_VEL
LIN {X 0,Y 178.552,Z 717.655,A -85,B 0,C 180,E1 9008.372,E2 9008.372} C_VEL
LIN {X 0,Y 178.343,Z 727.927,A -85,B 0,C 180,E1 9004.18,E2 9004.18} C_VEL
LIN {X 0,Y 178.815,Z 736.779,A -85,B 0,C 180,E1 8999.68,E2 8999.68} C_VEL
LIN {X 0,Y 180.206,Z 744.302,A -85,B 0,C 180,E1 8994.907,E2 8994.907} C_VEL
LIN {X 0,Y 183.087,Z 750.545,A -85,B 0,C 180,E1 8989.618,E2 8989.618} C_VEL
LIN {X 0,Y 187.179,Z 754.56,A -85,B 0,C 180,E1 8984.827,E2 8984.827} C_VEL
LIN {X 0,Y 192.985,Z 756.872,A -85,B 0,C 180,E1 8980.005,E2 8980.005} C_VEL
LIN {X 0,Y 200.251,Z 757.395,A -85,B 0,C 180,E1 8975.518,E2 8975.518} C_VEL
LIN {X 0,Y 208.861,Z 756.153,A -85,B 0,C 180,E1 8971.399,E2 8971.399} C_VEL
LIN {X 0,Y 219.868,Z 752.776,A -85,B 0,C 180,E1 8967.278,E2 8967.278} C_VEL
LIN {X 0,Y 231.074,Z 747.964,A -85,B 0,C 180,E1 8963.952,E2 8963.952} C_VEL
LIN {X 0,Y 236.817,Z 745.009,A -85,B 0,C 180,E1 8962.49,E2 8962.49} C_VEL
LIN {X 0,Y 236.867,Z 745.194,A -85,B 0,C 180,E1 8962.111,E2 8962.111} C_VEL
LIN {X 0,Y 235.337,Z 746.475,A -85,B 0,C 180,E1 8961.668,E2 8961.668} C_VEL
LIN {X 0,Y 231.73,Z 748.979,A -85,B 0,C 180,E1 8961.221,E2 8961.221} C_VEL
LIN {X 0,Y 222.426,Z 754.69,A -85,B 0,C 180,E1 8960.536,E2 8960.536} C_VEL
LIN {X 0,Y 218.716,Z 756.964,A -85,B 0,C 180,E1 8959.905,E2 8959.905} C_VEL
LIN {X 0,Y 204.256,Z 766.316,A -85,B 0,C 180,E1 8955.618,E2 8955.618} C_VEL
LIN {X 0,Y 191.572,Z 774.24,A -85,B 0,C 180,E1 8950.33,E2 8950.33} C_VEL
LIN {X 0,Y 181.536,Z 780.496,A -85,B 0,C 180,E1 8944.18,E2 8944.18} C_VEL
LIN {X 0,Y 174.54,Z 785.121,A -85,B 0,C 180,E1 8937.277,E2 8937.277} C_VEL
LIN {X 0,Y 170.899,Z 788.059,A -85,B 0,C 180,E1 8929.836,E2 8929.836} C_VEL
LIN {X 0,Y 170.688,Z 788.424,A -85,B 0,C 180,E1 8928.795,E2 8928.795} C_VEL
LIN {X 0,Y 169.51,Z 798.622,A -85,B 0,C 180,E1 8923.282,E2 8923.282} C_VEL
LIN {X 0,Y 169.293,Z 806.547,A -85,B 0,C 180,E1 8917.807,E2 8917.807} C_VEL
LIN {X 0,Y 169.537,Z 811.805,A -85,B 0,C 180,E1 8913.043,E2 8913.043} C_VEL
LIN {X 0,Y 169.448,Z 815.171,A -85,B 0,C 180,E1 8908.986,E2 8908.986} C_VEL
LIN {X 0,Y 168.799,Z 817.899,A -85,B 0,C 180,E1 8903.879,E2 8903.879} C_VEL
LIN {X 0,Y 168.795,Z 819.785,A -85,B 0,C 180,E1 8896.992,E2 8896.992} C_VEL
LIN {X 0,Y 171.242,Z 819.906,A -85,B 0,C 180,E1 8889.492,E2 8889.492} C_VEL
LIN {X 0,Y 176.956,Z 818.095,A -85,B 0,C 180,E1 8882.032,E2 8882.032} C_VEL
LIN {X 0,Y 186.326,Z 814.304,A -85,B 0,C 180,E1 8874.957,E2 8874.957} C_VEL
LIN {X 0,Y 198.852,Z 808.741,A -85,B 0,C 180,E1 8868.8,E2 8868.8} C_VEL
LIN {X 0,Y 214.12,Z 801.536,A -85,B 0,C 180,E1 8863.631,E2 8863.631} C_VEL
LIN {X 0,Y 216.927,Z 800.192,A -85,B 0,C 180,E1 8862.811,E2 8862.811} C_VEL
LIN {X 0,Y 202.232,Z 804.835,A -85,B 0,C 180,E1 8857.812,E2 8857.812} C_VEL
LIN {X 0,Y 190.131,Z 807.679,A -85,B 0,C 180,E1 8852.082,E2 8852.082} C_VEL
LIN {X 0,Y 180.617,Z 808.736,A -85,B 0,C 180,E1 8845.581,E2 8845.581} C_VEL
LIN {X 0,Y 174.142,Z 807.962,A -85,B 0,C 180,E1 8838.755,E2 8838.755} C_VEL
LIN {X 0,Y 170.372,Z 805.461,A -85,B 0,C 180,E1 8831.853,E2 8831.853} C_VEL
LIN {X 0,Y 168.766,Z 801.571,A -85,B 0,C 180,E1 8825.439,E2 8825.439} C_VEL
LIN {X 0,Y 168.338,Z 796.607,A -85,B 0,C 180,E1 8819.659,E2 8819.659} C_VEL
LIN {X 0,Y 168.391,Z 790.44,A -85,B 0,C 180,E1 8814.206,E2 8814.206} C_VEL
LIN {X 0,Y 168.982,Z 782.579,A -85,B 0,C 180,E1 8808.74,E2 8808.74} C_VEL
LIN {X 0,Y 170.362,Z 772.767,A -85,B 0,C 180,E1 8803.286,E2 8803.286} C_VEL
LIN {X 0,Y 172.732,Z 760.685,A -85,B 0,C 180,E1 8797.898,E2 8797.898} C_VEL
LIN {X 0,Y 175.817,Z 747.437,A -85,B 0,C 180,E1 8793.12,E2 8793.12} C_VEL
LIN {X 0,Y 179.516,Z 732.649,A -85,B 0,C 180,E1 8788.802,E2 8788.802} C_VEL
LIN {X 0,Y 183.739,Z 715.826,A -85,B 0,C 180,E1 8784.869,E2 8784.869} C_VEL
LIN {X 0,Y 188.038,Z 697.907,A -85,B 0,C 180,E1 8781.528,E2 8781.528} C_VEL
LIN {X 0,Y 192.302,Z 678.539,A -85,B 0,C 180,E1 8778.675,E2 8778.675} C_VEL
LIN {X 0,Y 196.001,Z 659.18,A -85,B 0,C 180,E1 8776.474,E2 8776.474} C_VEL
LIN {X 0,Y 199.446,Z 637.224,A -85,B 0,C 180,E1 8774.6,E2 8774.6} C_VEL
LIN {X 0,Y 202.652,Z 610.579,A -85,B 0,C 180,E1 8773.009,E2 8773.009} C_VEL
LIN {X 0,Y 216.74,Z 494.837,A -85,B 0,C 180,E1 8767.139,E2 8767.139} C_VEL
LIN {X 0,Y 205.432,Z 470.38,A -85,B 0,C 180,E1 8763.168,E2 8763.168} C_VEL
LIN {X 0,Y 194.806,Z 449.301,A -85,B 0,C 180,E1 8759.057,E2 8759.057} C_VEL
LIN {X 0,Y 184.69,Z 431.046,A -85,B 0,C 180,E1 8754.764,E2 8754.764} C_VEL
LIN {X 0,Y 179.422,Z 422.131,A -85,B 0,C 180,E1 8752.268,E2 8752.268} C_VEL
LIN {X 0,Y 175.218,Z 413.861,A -85,B 0,C 180,E1 8748.982,E2 8748.982} C_VEL
LIN {X 0,Y 173.427,Z 410.057,A -85,B 0,C 180,E1 8747.445,E2 8747.445} C_VEL
LIN {X 0,Y 171.483,Z 406.706,A -85,B 0,C 180,E1 8745.905,E2 8745.905} C_VEL
LIN {X 0,Y 171.217,Z 405.474,A -85,B 0,C 180,E1 8745.426,E2 8745.426} C_VEL
LIN {X 0,Y 171.216,Z 405.462,A -85,B 0,C 180,E1 8739.411,E2 8739.411} C_VEL
LIN {X 0,Y 171.219,Z 405.456,A -85,B 0,C 180,E1 8733.683,E2 8733.683} C_VEL
LIN {X 0,Y 171.221,Z 405.454,A -85,B 0,C 180,E1 8727.657,E2 8727.657} C_VEL
LIN {X 0,Y 171.226,Z 405.459,A -85,B 0,C 180,E1 8721.606,E2 8721.606} C_VEL
LIN {X 0,Y 171.227,Z 405.473,A -85,B 0,C 180,E1 8715.458,E2 8715.458} C_VEL
LIN {X 0,Y 171.226,Z 405.466,A -85,B 0,C 180,E1 8709.49,E2 8709.49} C_VEL
LIN {X 0,Y 171.249,Z 405.704,A -85,B 0,C 180,E1 8706.761,E2 8706.761} C_VEL
LIN {X 0,Y 174.498,Z 415.183,A -85,B 0,C 180,E1 8701.602,E2 8701.602} C_VEL
LIN {X 0,Y 177.784,Z 425.503,A -85,B 0,C 180,E1 8696.554,E2 8696.554} C_VEL
LIN {X 0,Y 181.141,Z 437.169,A -85,B 0,C 180,E1 8691.41,E2 8691.41} C_VEL
LIN {X 0,Y 184.524,Z 450.448,A -85,B 0,C 180,E1 8686.11,E2 8686.11} C_VEL
LIN {X 0,Y 187.779,Z 464.815,A -85,B 0,C 180,E1 8680.878,E2 8680.878} C_VEL
LIN {X 0,Y 188.213,Z 467.401,A -85,B 0,C 180,E1 8680.001,E2 8680.001} C_VEL
LIN {X 0,Y 186.029,Z 475.449,A -85,B 0,C 180,E1 8677.831,E2 8677.831} C_VEL
LIN {X 0,Y 186.834,Z 505.599,A -85,B 0,C 180,E1 8675.488,E2 8675.488} C_VEL
LIN {X 0,Y 187.916,Z 525.964,A -85,B 0,C 180,E1 8673.873,E2 8673.873} C_VEL
LIN {X 0,Y 180.071,Z 617.674,A -85,B 0,C 180,E1 8667.656,E2 8667.656} C_VEL
LIN {X 0,Y 178.352,Z 638.115,A -85,B 0,C 180,E1 8665.663,E2 8665.663} C_VEL
LIN {X 0,Y 176.421,Z 656.631,A -85,B 0,C 180,E1 8663.197,E2 8663.197} C_VEL
LIN {X 0,Y 174.476,Z 674.436,A -85,B 0,C 180,E1 8660.111,E2 8660.111} C_VEL
LIN {X 0,Y 172.692,Z 690.876,A -85,B 0,C 180,E1 8656.482,E2 8656.482} C_VEL
LIN {X 0,Y 171.297,Z 705.798,A -85,B 0,C 180,E1 8652.302,E2 8652.302} C_VEL
LIN {X 0,Y 170.528,Z 717.993,A -85,B 0,C 180,E1 8648.09,E2 8648.09} C_VEL
LIN {X 0,Y 170.367,Z 728.406,A -85,B 0,C 180,E1 8643.702,E2 8643.702} C_VEL
LIN {X 0,Y 171.006,Z 738.007,A -85,B 0,C 180,E1 8638.66,E2 8638.66} C_VEL
LIN {X 0,Y 172.795,Z 745.988,A -85,B 0,C 180,E1 8633.355,E2 8633.355} C_VEL
LIN {X 0,Y 176.165,Z 752.213,A -85,B 0,C 180,E1 8627.878,E2 8627.878} C_VEL
LIN {X 0,Y 180.805,Z 756.252,A -85,B 0,C 180,E1 8622.957,E2 8622.957} C_VEL
LIN {X 0,Y 187.251,Z 758.64,A -85,B 0,C 180,E1 8618.052,E2 8618.052} C_VEL
LIN {X 0,Y 195.698,Z 759.275,A -85,B 0,C 180,E1 8613.282,E2 8613.282} C_VEL
LIN {X 0,Y 205.646,Z 757.979,A -85,B 0,C 180,E1 8608.978,E2 8608.978} C_VEL
LIN {X 0,Y 216.97,Z 754.862,A -85,B 0,C 180,E1 8605.151,E2 8605.151} C_VEL
LIN {X 0,Y 228.168,Z 750.594,A -85,B 0,C 180,E1 8602.072,E2 8602.072} C_VEL
LIN {X 0,Y 218.716,Z 756.964,A -85,B 0,C 180,E1 8599.905,E2 8599.905} C_VEL
LIN {X 0,Y 213.087,Z 760.379,A -85,B 0,C 180,E1 8598.786,E2 8598.786} C_VEL
LIN {X 0,Y 198.69,Z 767.319,A -85,B 0,C 180,E1 8596.566,E2 8596.566} C_VEL
LIN {X 0,Y 193.12,Z 769.912,A -85,B 0,C 180,E1 8595.205,E2 8595.205} C_VEL
LIN {X 0,Y 191.788,Z 770.579,A -85,B 0,C 180,E1 8594.725,E2 8594.725} C_VEL
LIN {X 0,Y 179.32,Z 777.269,A -85,B 0,C 180,E1 8588.645,E2 8588.645} C_VEL
LIN {X 0,Y 170.003,Z 782.286,A -85,B 0,C 180,E1 8581.564,E2 8581.564} C_VEL
LIN {X 0,Y 164.488,Z 785.458,A -85,B 0,C 180,E1 8574.034,E2 8574.034} C_VEL
LIN {X 0,Y 162.847,Z 786.908,A -85,B 0,C 180,E1 8568.991,E2 8568.991} C_VEL
LIN {X 0,Y 161.674,Z 796.632,A -85,B 0,C 180,E1 8563.592,E2 8563.592} C_VEL
LIN {X 0,Y 161.424,Z 804.387,A -85,B 0,C 180,E1 8558.19,E2 8558.19} C_VEL
LIN {X 0,Y 161.683,Z 809.992,A -85,B 0,C 180,E1 8553.191,E2 8553.191} C_VEL
LIN {X 0,Y 161.618,Z 813.536,A -85,B 0,C 180,E1 8548.937,E2 8548.937} C_VEL
LIN {X 0,Y 160.907,Z 816.558,A -85,B 0,C 180,E1 8543.578,E2 8543.578} C_VEL
LIN {X 0,Y 160.956,Z 818.764,A -85,B 0,C 180,E1 8536.346,E2 8536.346} C_VEL
LIN {X 0,Y 163.666,Z 819.265,A -85,B 0,C 180,E1 8528.497,E2 8528.497} C_VEL
LIN {X 0,Y 169.833,Z 817.913,A -85,B 0,C 180,E1 8520.748,E2 8520.748} C_VEL
LIN {X 0,Y 179.79,Z 814.667,A -85,B 0,C 180,E1 8513.483,E2 8513.483} C_VEL
LIN {X 0,Y 192.937,Z 809.727,A -85,B 0,C 180,E1 8507.243,E2 8507.243} C_VEL
LIN {X 0,Y 206.342,Z 804.217,A -85,B 0,C 180,E1 8502.718,E2 8502.718} C_VEL
LIN {X 0,Y 191.471,Z 807.735,A -85,B 0,C 180,E1 8497.283,E2 8497.283} C_VEL
LIN {X 0,Y 179.679,Z 809.403,A -85,B 0,C 180,E1 8491.166,E2 8491.166} C_VEL
LIN {X 0,Y 170.956,Z 809.338,A -85,B 0,C 180,E1 8484.535,E2 8484.535} C_VEL
LIN {X 0,Y 164.945,Z 807.521,A -85,B 0,C 180,E1 8477.279,E2 8477.279} C_VEL
LIN {X 0,Y 161.705,Z 804.011,A -85,B 0,C 180,E1 8469.969,E2 8469.969} C_VEL
LIN {X 0,Y 160.536,Z 799.147,A -85,B 0,C 180,E1 8463.213,E2 8463.213} C_VEL
LIN {X 0,Y 160.338,Z 793.582,A -85,B 0,C 180,E1 8457.498,E2 8457.498} C_VEL
LIN {X 0,Y 160.607,Z 786.458,A -85,B 0,C 180,E1 8451.767,E2 8451.767} C_VEL
LIN {X 0,Y 161.555,Z 777.5,A -85,B 0,C 180,E1 8446.032,E2 8446.032} C_VEL
LIN {X 0,Y 163.468,Z 766.43,A -85,B 0,C 180,E1 8440.341,E2 8440.341} C_VEL
LIN {X 0,Y 166.26,Z 753.827,A -85,B 0,C 180,E1 8435.104,E2 8435.104} C_VEL
LIN {X 0,Y 169.798,Z 739.66,A -85,B 0,C 180,E1 8430.354,E2 8430.354} C_VEL
LIN {X 0,Y 173.885,Z 723.853,A -85,B 0,C 180,E1 8426.098,E2 8426.098} C_VEL
LIN {X 0,Y 178.328,Z 706.322,A -85,B 0,C 180,E1 8422.327,E2 8422.327} C_VEL
LIN {X 0,Y 182.694,Z 687.947,A -85,B 0,C 180,E1 8419.19,E2 8419.19} C_VEL
LIN {X 0,Y 186.639,Z 669.45,A -85,B 0,C 180,E1 8416.707,E2 8416.707} C_VEL
LIN {X 0,Y 190.444,Z 648.331,A -85,B 0,C 180,E1 8414.544,E2 8414.544} C_VEL
LIN {X 0,Y 193.562,Z 626.629,A -85,B 0,C 180,E1 8412.927,E2 8412.927} C_VEL
LIN {X 0,Y 209.818,Z 497.258,A -85,B 0,C 180,E1 8406.053,E2 8406.053} C_VEL
LIN {X 0,Y 199.177,Z 473.953,A -85,B 0,C 180,E1 8402.106,E2 8402.106} C_VEL
LIN {X 0,Y 188.94,Z 453.557,A -85,B 0,C 180,E1 8397.969,E2 8397.969} C_VEL
LIN {X 0,Y 179.516,Z 436.31,A -85,B 0,C 180,E1 8393.773,E2 8393.773} C_VEL
LIN {X 0,Y 171.536,Z 422.996,A -85,B 0,C 180,E1 8389.848,E2 8389.848} C_VEL
LIN {X 0,Y 167.724,Z 415.387,A -85,B 0,C 180,E1 8386.627,E2 8386.627} C_VEL
LIN {X 0,Y 165.215,Z 410.747,A -85,B 0,C 180,E1 8384.463,E2 8384.463} C_VEL
LIN {X 0,Y 163.607,Z 407.935,A -85,B 0,C 180,E1 8383.069,E2 8383.069} C_VEL
LIN {X 0,Y 163.283,Z 406.452,A -85,B 0,C 180,E1 8382.466,E2 8382.466} C_VEL
LIN {X 0,Y 163.291,Z 406.459,A -85,B 0,C 180,E1 8376.328,E2 8376.328} C_VEL
LIN {X 0,Y 163.297,Z 406.452,A -85,B 0,C 180,E1 8370,E2 8370} C_VEL
LIN {X 0,Y 163.289,Z 406.452,A -85,B 0,C 180,E1 8363.672,E2 8363.672} C_VEL
LIN {X 0,Y 163.283,Z 406.451,A -85,B 0,C 180,E1 8357.624,E2 8357.624} C_VEL
LIN {X 0,Y 163.285,Z 406.462,A -85,B 0,C 180,E1 8351.433,E2 8351.433} C_VEL
LIN {X 0,Y 163.301,Z 406.611,A -85,B 0,C 180,E1 8349.105,E2 8349.105} C_VEL
LIN {X 0,Y 166.577,Z 415.953,A -85,B 0,C 180,E1 8343.629,E2 8343.629} C_VEL
LIN {X 0,Y 170.007,Z 426.691,A -85,B 0,C 180,E1 8338.041,E2 8338.041} C_VEL
LIN {X 0,Y 173.302,Z 438.157,A -85,B 0,C 180,E1 8332.714,E2 8332.714} C_VEL
LIN {X 0,Y 176.633,Z 451.291,A -85,B 0,C 180,E1 8327.212,E2 8327.212} C_VEL
LIN {X 0,Y 179.821,Z 465.397,A -85,B 0,C 180,E1 8321.834,E2 8321.834} C_VEL
LIN {X 0,Y 180.461,Z 468.808,A -85,B 0,C 180,E1 8320.618,E2 8320.618} C_VEL
LIN {X 0,Y 178.622,Z 475.45,A -85,B 0,C 180,E1 8318.798,E2 8318.798} C_VEL
LIN {X 0,Y 179.245,Z 505.289,A -85,B 0,C 180,E1 8316.392,E2 8316.392} C_VEL
LIN {X 0,Y 180.289,Z 526.462,A -85,B 0,C 180,E1 8314.643,E2 8314.643} C_VEL
LIN {X 0,Y 172.027,Z 619.997,A -85,B 0,C 180,E1 8307.933,E2 8307.933} C_VEL
LIN {X 0,Y 170.33,Z 639.246,A -85,B 0,C 180,E1 8305.934,E2 8305.934} C_VEL
LIN {X 0,Y 168.294,Z 658.209,A -85,B 0,C 180,E1 8303.272,E2 8303.272} C_VEL
LIN {X 0,Y 166.339,Z 675.732,A -85,B 0,C 180,E1 8300.037,E2 8300.037} C_VEL
LIN {X 0,Y 164.486,Z 692.639,A -85,B 0,C 180,E1 8296.057,E2 8296.057} C_VEL
LIN {X 0,Y 163.143,Z 707.509,A -85,B 0,C 180,E1 8291.669,E2 8291.669} C_VEL
LIN {X 0,Y 162.482,Z 719.086,A -85,B 0,C 180,E1 8287.425,E2 8287.425} C_VEL
LIN {X 0,Y 162.451,Z 730.239,A -85,B 0,C 180,E1 8282.47,E2 8282.47} C_VEL
LIN {X 0,Y 163.442,Z 740.252,A -85,B 0,C 180,E1 8276.844,E2 8276.844} C_VEL
LIN {X 0,Y 165.528,Z 747.607,A -85,B 0,C 180,E1 8271.665,E2 8271.665} C_VEL
LIN {X 0,Y 169.147,Z 753.516,A -85,B 0,C 180,E1 8266.323,E2 8266.323} C_VEL
LIN {X 0,Y 174.656,Z 757.923,A -85,B 0,C 180,E1 8260.955,E2 8260.955} C_VEL
LIN {X 0,Y 181.773,Z 760.409,A -85,B 0,C 180,E1 8255.981,E2 8255.981} C_VEL
LIN {X 0,Y 190.946,Z 761.183,A -85,B 0,C 180,E1 8251.201,E2 8251.201} C_VEL
LIN {X 0,Y 201.63,Z 760.134,A -85,B 0,C 180,E1 8246.943,E2 8246.943} C_VEL
LIN {X 0,Y 214.355,Z 757.063,A -85,B 0,C 180,E1 8243.007,E2 8243.007} C_VEL
LIN {X 0,Y 216.946,Z 756.304,A -85,B 0,C 180,E1 8242.278,E2 8242.278} C_VEL
LIN {X 0,Y 202.076,Z 764.934,A -85,B 0,C 180,E1 8238.344,E2 8238.344} C_VEL
LIN {X 0,Y 191.788,Z 770.579,A -85,B 0,C 180,E1 8234.725,E2 8234.725} C_VEL
LIN {X 0,Y 186.299,Z 773.069,A -85,B 0,C 180,E1 8232.97,E2 8232.97} C_VEL
LIN {X 0,Y 172.679,Z 777.318,A -85,B 0,C 180,E1 8229.245,E2 8229.245} C_VEL
LIN {X 0,Y 168.181,Z 778.77,A -85,B 0,C 180,E1 8227.193,E2 8227.193} C_VEL
LIN {X 0,Y 167.695,Z 778.965,A -85,B 0,C 180,E1 8226.862,E2 8226.862} C_VEL
LIN {X 0,Y 159.661,Z 782.575,A -85,B 0,C 180,E1 8219.24,E2 8219.24} C_VEL
LIN {X 0,Y 155.423,Z 784.555,A -85,B 0,C 180,E1 8210.722,E2 8210.722} C_VEL
LIN {X 0,Y 155.116,Z 784.96,A -85,B 0,C 180,E1 8209.388,E2 8209.388} C_VEL
LIN {X 0,Y 153.803,Z 795.181,A -85,B 0,C 180,E1 8203.535,E2 8203.535} C_VEL
LIN {X 0,Y 153.597,Z 803.527,A -85,B 0,C 180,E1 8197.481,E2 8197.481} C_VEL
LIN {X 0,Y 153.884,Z 809.121,A -85,B 0,C 180,E1 8192.234,E2 8192.234} C_VEL
LIN {X 0,Y 153.705,Z 812.338,A -85,B 0,C 180,E1 8188.136,E2 8188.136} C_VEL
LIN {X 0,Y 152.963,Z 815.4,A -85,B 0,C 180,E1 8182.488,E2 8182.488} C_VEL
LIN {X 0,Y 153.314,Z 817.713,A -85,B 0,C 180,E1 8174.839,E2 8174.839} C_VEL
LIN {X 0,Y 156.597,Z 818.417,A -85,B 0,C 180,E1 8166.68,E2 8166.68} C_VEL
LIN {X 0,Y 163.554,Z 817.366,A -85,B 0,C 180,E1 8158.692,E2 8158.692} C_VEL
LIN {X 0,Y 174.405,Z 814.519,A -85,B 0,C 180,E1 8151.325,E2 8151.325} C_VEL
LIN {X 0,Y 189.077,Z 809.849,A -85,B 0,C 180,E1 8144.878,E2 8144.878} C_VEL
LIN {X 0,Y 195.772,Z 807.536,A -85,B 0,C 180,E1 8142.655,E2 8142.655} C_VEL
LIN {X 0,Y 181.257,Z 809.852,A -85,B 0,C 180,E1 8136.96,E2 8136.96} C_VEL
LIN {X 0,Y 169.698,Z 810.44,A -85,B 0,C 180,E1 8130.445,E2 8130.445} C_VEL
LIN {X 0,Y 161.037,Z 809.263,A -85,B 0,C 180,E1 8123.026,E2 8123.026} C_VEL
LIN {X 0,Y 155.676,Z 806.312,A -85,B 0,C 180,E1 8115.267,E2 8115.267} C_VEL
LIN {X 0,Y 153.184,Z 801.945,A -85,B 0,C 180,E1 8107.878,E2 8107.878} C_VEL
LIN {X 0,Y 152.453,Z 796.421,A -85,B 0,C 180,E1 8101.127,E2 8101.127} C_VEL
LIN {X 0,Y 152.425,Z 789.953,A -85,B 0,C 180,E1 8095.108,E2 8095.108} C_VEL
LIN {X 0,Y 152.978,Z 781.786,A -85,B 0,C 180,E1 8089.073,E2 8089.073} C_VEL
LIN {X 0,Y 154.292,Z 772.334,A -85,B 0,C 180,E1 8083.433,E2 8083.433} C_VEL
LIN {X 0,Y 156.611,Z 760.692,A -85,B 0,C 180,E1 8077.78,E2 8077.78} C_VEL
LIN {X 0,Y 159.906,Z 747.065,A -85,B 0,C 180,E1 8072.438,E2 8072.438} C_VEL
LIN {X 0,Y 164.005,Z 731.432,A -85,B 0,C 180,E1 8067.554,E2 8067.554} C_VEL
LIN {X 0,Y 168.452,Z 714.658,A -85,B 0,C 180,E1 8063.378,E2 8063.378} C_VEL
LIN {X 0,Y 173.169,Z 696.056,A -85,B 0,C 180,E1 8059.708,E2 8059.708} C_VEL
LIN {X 0,Y 177.513,Z 677.243,A -85,B 0,C 180,E1 8056.814,E2 8056.814} C_VEL
LIN {X 0,Y 181.589,Z 656.901,A -85,B 0,C 180,E1 8054.403,E2 8054.403} C_VEL
LIN {X 0,Y 185.113,Z 635.441,A -85,B 0,C 180,E1 8052.507,E2 8052.507} C_VEL
LIN {X 0,Y 196.214,Z 549.278,A -85,B 0,C 180,E1 8047.485,E2 8047.485} C_VEL
LIN {X 0,Y 202.915,Z 499.573,A -85,B 0,C 180,E1 8044.908,E2 8044.908} C_VEL
LIN {X 0,Y 192.377,Z 476.414,A -85,B 0,C 180,E1 8040.794,E2 8040.794} C_VEL
LIN {X 0,Y 182.073,Z 455.732,A -85,B 0,C 180,E1 8036.368,E2 8036.368} C_VEL
LIN {X 0,Y 172.347,Z 437.988,A -85,B 0,C 180,E1 8031.738,E2 8031.738} C_VEL
LIN {X 0,Y 164.282,Z 424.719,A -85,B 0,C 180,E1 8027.488,E2 8027.488} C_VEL
LIN {X 0,Y 160.315,Z 416.974,A -85,B 0,C 180,E1 8024.078,E2 8024.078} C_VEL
LIN {X 0,Y 158.115,Z 412.992,A -85,B 0,C 180,E1 8022.045,E2 8022.045} C_VEL
LIN {X 0,Y 155.817,Z 409.327,A -85,B 0,C 180,E1 8019.977,E2 8019.977} C_VEL
LIN {X 0,Y 155.337,Z 407.438,A -85,B 0,C 180,E1 8019.073,E2 8019.073} C_VEL
LIN {X 0,Y 155.335,Z 407.436,A -85,B 0,C 180,E1 8012.952,E2 8012.952} C_VEL
LIN {X 0,Y 155.335,Z 407.434,A -85,B 0,C 180,E1 8007.048,E2 8007.048} C_VEL
LIN {X 0,Y 155.337,Z 407.443,A -85,B 0,C 180,E1 8000.74,E2 8000.74} C_VEL
LIN {X 0,Y 155.341,Z 407.448,A -85,B 0,C 180,E1 7994.316,E2 7994.316} C_VEL
LIN {X 0,Y 155.378,Z 407.658,A -85,B 0,C 180,E1 7991.62,E2 7991.62} C_VEL
LIN {X 0,Y 158.647,Z 416.795,A -85,B 0,C 180,E1 7985.817,E2 7985.817} C_VEL
LIN {X 0,Y 162.005,Z 427.192,A -85,B 0,C 180,E1 7980.005,E2 7980.005} C_VEL
LIN {X 0,Y 165.232,Z 438.335,A -85,B 0,C 180,E1 7974.484,E2 7974.484} C_VEL
LIN {X 0,Y 168.434,Z 450.828,A -85,B 0,C 180,E1 7968.93,E2 7968.93} C_VEL
LIN {X 0,Y 171.395,Z 463.828,A -85,B 0,C 180,E1 7963.666,E2 7963.666} C_VEL
LIN {X 0,Y 172.724,Z 470.083,A -85,B 0,C 180,E1 7961.294,E2 7961.294} C_VEL
LIN {X 0,Y 171.226,Z 475.33,A -85,B 0,C 180,E1 7959.817,E2 7959.817} C_VEL
LIN {X 0,Y 171.638,Z 504.729,A -85,B 0,C 180,E1 7957.342,E2 7957.342} C_VEL
LIN {X 0,Y 172.632,Z 526.942,A -85,B 0,C 180,E1 7955.419,E2 7955.419} C_VEL
LIN {X 0,Y 164.119,Z 620.607,A -85,B 0,C 180,E1 7948.387,E2 7948.387} C_VEL
LIN {X 0,Y 162.39,Z 639.472,A -85,B 0,C 180,E1 7946.316,E2 7946.316} C_VEL
LIN {X 0,Y 160.304,Z 658.349,A -85,B 0,C 180,E1 7943.525,E2 7943.525} C_VEL
LIN {X 0,Y 158.209,Z 676.805,A -85,B 0,C 180,E1 7939.955,E2 7939.955} C_VEL
LIN {X 0,Y 156.416,Z 693.089,A -85,B 0,C 180,E1 7935.955,E2 7935.955} C_VEL
LIN {X 0,Y 155.092,Z 707.926,A -85,B 0,C 180,E1 7931.34,E2 7931.34} C_VEL
LIN {X 0,Y 154.457,Z 720.096,A -85,B 0,C 180,E1 7926.692,E2 7926.692} C_VEL
LIN {X 0,Y 154.56,Z 731.205,A -85,B 0,C 180,E1 7921.483,E2 7921.483} C_VEL
LIN {X 0,Y 155.561,Z 740.153,A -85,B 0,C 180,E1 7916.315,E2 7916.315} C_VEL
LIN {X 0,Y 157.998,Z 748.301,A -85,B 0,C 180,E1 7910.53,E2 7910.53} C_VEL
LIN {X 0,Y 161.974,Z 754.475,A -85,B 0,C 180,E1 7904.974,E2 7904.974} C_VEL
LIN {X 0,Y 168.338,Z 759.335,A -85,B 0,C 180,E1 7899.123,E2 7899.123} C_VEL
LIN {X 0,Y 176.069,Z 762.096,A -85,B 0,C 180,E1 7894.071,E2 7894.071} C_VEL
LIN {X 0,Y 185.894,Z 763.109,A -85,B 0,C 180,E1 7889.272,E2 7889.272} C_VEL
LIN {X 0,Y 197.229,Z 762.381,A -85,B 0,C 180,E1 7885.051,E2 7885.051} C_VEL
LIN {X 0,Y 205.573,Z 760.959,A -85,B 0,C 180,E1 7882.448,E2 7882.448} C_VEL
LIN {X 0,Y 190.02,Z 768.676,A -85,B 0,C 180,E1 7877.896,E2 7877.896} C_VEL
LIN {X 0,Y 176.716,Z 774.888,A -85,B 0,C 180,E1 7872.323,E2 7872.323} C_VEL
LIN {X 0,Y 167.695,Z 778.965,A -85,B 0,C 180,E1 7866.862,E2 7866.862} C_VEL
LIN {X 0,Y 163.421,Z 780.299,A -85,B 0,C 180,E1 7864.425,E2 7864.425} C_VEL
LIN {X 0,Y 152.373,Z 781.653,A -85,B 0,C 180,E1 7858.832,E2 7858.832} C_VEL
LIN {X 0,Y 149.596,Z 781.979,A -85,B 0,C 180,E1 7856.092,E2 7856.092} C_VEL
LIN {X 0,Y 149.485,Z 782.004,A -85,B 0,C 180,E1 7855.885,E2 7855.885} C_VEL
LIN {X 0,Y 147.472,Z 782.766,A -85,B 0,C 180,E1 7849.919,E2 7849.919} C_VEL
LIN {X 0,Y 145.943,Z 793.656,A -85,B 0,C 180,E1 7843.47,E2 7843.47} C_VEL
LIN {X 0,Y 145.76,Z 801.686,A -85,B 0,C 180,E1 7837.489,E2 7837.489} C_VEL
LIN {X 0,Y 146.081,Z 807.098,A -85,B 0,C 180,E1 7832.354,E2 7832.354} C_VEL
LIN {X 0,Y 145.904,Z 810.567,A -85,B 0,C 180,E1 7828.036,E2 7828.036} C_VEL
LIN {X 0,Y 145.093,Z 813.969,A -85,B 0,C 180,E1 7821.679,E2 7821.679} C_VEL
LIN {X 0,Y 145.767,Z 816.605,A -85,B 0,C 180,E1 7813.256,E2 7813.256} C_VEL
LIN {X 0,Y 149.969,Z 817.548,A -85,B 0,C 180,E1 7804.319,E2 7804.319} C_VEL
LIN {X 0,Y 157.932,Z 816.748,A -85,B 0,C 180,E1 7796.143,E2 7796.143} C_VEL
LIN {X 0,Y 169.858,Z 814.252,A -85,B 0,C 180,E1 7788.755,E2 7788.755} C_VEL
LIN {X 0,Y 185.067,Z 810.17,A -85,B 0,C 180,E1 7782.537,E2 7782.537} C_VEL
LIN {X 0,Y 170.474,Z 811.333,A -85,B 0,C 180,E1 7776.326,E2 7776.326} C_VEL
LIN {X 0,Y 159.31,Z 810.768,A -85,B 0,C 180,E1 7769.31,E2 7769.31} C_VEL
LIN {X 0,Y 151.525,Z 808.566,A -85,B 0,C 180,E1 7761.686,E2 7761.686} C_VEL
LIN {X 0,Y 146.759,Z 804.574,A -85,B 0,C 180,E1 7753.393,E2 7753.393} C_VEL
LIN {X 0,Y 144.891,Z 799.531,A -85,B 0,C 180,E1 7745.941,E2 7745.941} C_VEL
LIN {X 0,Y 144.455,Z 793.885,A -85,B 0,C 180,E1 7739.603,E2 7739.603} C_VEL
LIN {X 0,Y 144.577,Z 786.665,A -85,B 0,C 180,E1 7733.248,E2 7733.248} C_VEL
LIN {X 0,Y 145.41,Z 777.626,A -85,B 0,C 180,E1 7726.884,E2 7726.884} C_VEL
LIN {X 0,Y 147.291,Z 766.467,A -85,B 0,C 180,E1 7720.571,E2 7720.571} C_VEL
LIN {X 0,Y 150.17,Z 753.762,A -85,B 0,C 180,E1 7714.778,E2 7714.778} C_VEL
LIN {X 0,Y 154.047,Z 738.874,A -85,B 0,C 180,E1 7709.368,E2 7709.368} C_VEL
LIN {X 0,Y 158.458,Z 722.717,A -85,B 0,C 180,E1 7704.687,E2 7704.687} C_VEL
LIN {X 0,Y 163.182,Z 705.11,A -85,B 0,C 180,E1 7700.641,E2 7700.641} C_VEL
LIN {X 0,Y 167.906,Z 686.248,A -85,B 0,C 180,E1 7697.245,E2 7697.245} C_VEL
LIN {X 0,Y 172.348,Z 666.256,A -85,B 0,C 180,E1 7694.473,E2 7694.473} C_VEL
LIN {X 0,Y 176.303,Z 645.178,A -85,B 0,C 180,E1 7692.26,E2 7692.26} C_VEL
LIN {X 0,Y 179.638,Z 622.35,A -85,B 0,C 180,E1 7690.557,E2 7690.557} C_VEL
LIN {X 0,Y 196.01,Z 501.806,A -85,B 0,C 180,E1 7683.693,E2 7683.693} C_VEL
LIN {X 0,Y 185.588,Z 478.82,A -85,B 0,C 180,E1 7679.402,E2 7679.402} C_VEL
LIN {X 0,Y 175.932,Z 459.338,A -85,B 0,C 180,E1 7675.005,E2 7675.005} C_VEL
LIN {X 0,Y 167.195,Z 443.197,A -85,B 0,C 180,E1 7670.615,E2 7670.615} C_VEL
LIN {X 0,Y 159.438,Z 430.197,A -85,B 0,C 180,E1 7666.307,E2 7666.307} C_VEL
LIN {X 0,Y 155.432,Z 423.654,A -85,B 0,C 180,E1 7663.769,E2 7663.769} C_VEL
LIN {X 0,Y 152.137,Z 417.621,A -85,B 0,C 180,E1 7660.604,E2 7660.604} C_VEL
LIN {X 0,Y 149.688,Z 413.085,A -85,B 0,C 180,E1 7658.064,E2 7658.064} C_VEL
LIN {X 0,Y 147.844,Z 410.213,A -85,B 0,C 180,E1 7656.212,E2 7656.212} C_VEL
LIN {X 0,Y 147.4,Z 408.43,A -85,B 0,C 180,E1 7655.352,E2 7655.352} C_VEL
LIN {X 0,Y 147.399,Z 408.422,A -85,B 0,C 180,E1 7648.834,E2 7648.834} C_VEL
LIN {X 0,Y 147.407,Z 408.423,A -85,B 0,C 180,E1 7642.203,E2 7642.203} C_VEL
LIN {X 0,Y 147.41,Z 408.439,A -85,B 0,C 180,E1 7635.465,E2 7635.465} C_VEL
LIN {X 0,Y 147.435,Z 408.681,A -85,B 0,C 180,E1 7634.462,E2 7634.462} C_VEL
LIN {X 0,Y 150.062,Z 416.007,A -85,B 0,C 180,E1 7629.32,E2 7629.32} C_VEL
LIN {X 0,Y 152.961,Z 424.458,A -85,B 0,C 180,E1 7624.026,E2 7624.026} C_VEL
LIN {X 0,Y 156.124,Z 434.768,A -85,B 0,C 180,E1 7618.321,E2 7618.321} C_VEL
LIN {X 0,Y 159.31,Z 446.609,A -85,B 0,C 180,E1 7612.497,E2 7612.497} C_VEL
LIN {X 0,Y 162.344,Z 459.329,A -85,B 0,C 180,E1 7606.871,E2 7606.871} C_VEL
LIN {X 0,Y 164.932,Z 471.522,A -85,B 0,C 180,E1 7601.953,E2 7601.953} C_VEL
LIN {X 0,Y 163.875,Z 475.197,A -85,B 0,C 180,E1 7600.913,E2 7600.913} C_VEL
LIN {X 0,Y 164.086,Z 504.118,A -85,B 0,C 180,E1 7598.383,E2 7598.383} C_VEL
LIN {X 0,Y 165.018,Z 527.297,A -85,B 0,C 180,E1 7596.27,E2 7596.27} C_VEL
LIN {X 0,Y 156.241,Z 620.4,A -85,B 0,C 180,E1 7588.879,E2 7588.879} C_VEL
LIN {X 0,Y 154.333,Z 640.619,A -85,B 0,C 180,E1 7586.553,E2 7586.553} C_VEL
LIN {X 0,Y 152.203,Z 659.418,A -85,B 0,C 180,E1 7583.624,E2 7583.624} C_VEL
LIN {X 0,Y 150.173,Z 677.021,A -85,B 0,C 180,E1 7580.054,E2 7580.054} C_VEL
LIN {X 0,Y 148.296,Z 693.926,A -85,B 0,C 180,E1 7575.646,E2 7575.646} C_VEL
LIN {X 0,Y 146.974,Z 709.365,A -85,B 0,C 180,E1 7570.585,E2 7570.585} C_VEL
LIN {X 0,Y 146.455,Z 721.792,A -85,B 0,C 180,E1 7565.485,E2 7565.485} C_VEL
LIN {X 0,Y 146.712,Z 732.084,A -85,B 0,C 180,E1 7560.391,E2 7560.391} C_VEL
LIN {X 0,Y 148.076,Z 741.695,A -85,B 0,C 180,E1 7554.576,E2 7554.576} C_VEL
LIN {X 0,Y 151.225,Z 750.266,A -85,B 0,C 180,E1 7548.173,E2 7548.173} C_VEL
LIN {X 0,Y 156.252,Z 756.644,A -85,B 0,C 180,E1 7542.113,E2 7542.113} C_VEL
LIN {X 0,Y 163.566,Z 761.396,A -85,B 0,C 180,E1 7536.206,E2 7536.206} C_VEL
LIN {X 0,Y 172.209,Z 764.052,A -85,B 0,C 180,E1 7531.191,E2 7531.191} C_VEL
LIN {X 0,Y 182.972,Z 765.072,A -85,B 0,C 180,E1 7526.502,E2 7526.502} C_VEL
LIN {X 0,Y 194.284,Z 764.545,A -85,B 0,C 180,E1 7522.614,E2 7522.614} C_VEL
LIN {X 0,Y 178.736,Z 771.065,A -85,B 0,C 180,E1 7517.597,E2 7517.597} C_VEL
LIN {X 0,Y 165.366,Z 776.275,A -85,B 0,C 180,E1 7511.228,E2 7511.228} C_VEL
LIN {X 0,Y 155.266,Z 779.99,A -85,B 0,C 180,E1 7503.629,E2 7503.629} C_VEL
LIN {X 0,Y 149.485,Z 782.004,A -85,B 0,C 180,E1 7495.885,E2 7495.885} C_VEL
LIN {X 0,Y 147.598,Z 782.102,A -85,B 0,C 180,E1 7493.939,E2 7493.939} C_VEL
LIN {X 0,Y 142.49,Z 782.486,A -85,B 0,C 180,E1 7490.856,E2 7490.856} C_VEL
LIN {X 0,Y 139.598,Z 783.92,A -85,B 0,C 180,E1 7488.771,E2 7488.771} C_VEL
LIN {X 0,Y 138.742,Z 785.669,A -85,B 0,C 180,E1 7487.465,E2 7487.465} C_VEL
LIN {X 0,Y 137.953,Z 794.945,A -85,B 0,C 180,E1 7481.285,E2 7481.285} C_VEL
LIN {X 0,Y 138.106,Z 802.474,A -85,B 0,C 180,E1 7474.984,E2 7474.984} C_VEL
LIN {X 0,Y 138.332,Z 807.116,A -85,B 0,C 180,E1 7470,E2 7470} C_VEL
LIN {X 0,Y 137.707,Z 810.424,A -85,B 0,C 180,E1 7465.002,E2 7465.002} C_VEL
LIN {X 0,Y 137.298,Z 813.935,A -85,B 0,C 180,E1 7456.953,E2 7456.953} C_VEL
LIN {X 0,Y 139.82,Z 816.113,A -85,B 0,C 180,E1 7447.728,E2 7447.728} C_VEL
LIN {X 0,Y 146.553,Z 816.599,A -85,B 0,C 180,E1 7438.518,E2 7438.518} C_VEL
LIN {X 0,Y 157.683,Z 815.34,A -85,B 0,C 180,E1 7430.176,E2 7430.176} C_VEL
LIN {X 0,Y 172.703,Z 812.404,A -85,B 0,C 180,E1 7423.157,E2 7423.157} C_VEL
LIN {X 0,Y 174.375,Z 812.013,A -85,B 0,C 180,E1 7422.442,E2 7422.442} C_VEL
LIN {X 0,Y 160.238,Z 812.068,A -85,B 0,C 180,E1 7415.912,E2 7415.912} C_VEL
LIN {X 0,Y 149.403,Z 810.458,A -85,B 0,C 180,E1 7408.369,E2 7408.369} C_VEL
LIN {X 0,Y 141.871,Z 807.061,A -85,B 0,C 180,E1 7399.772,E2 7399.772} C_VEL
LIN {X 0,Y 137.902,Z 801.948,A -85,B 0,C 180,E1 7390.865,E2 7390.865} C_VEL
LIN {X 0,Y 136.672,Z 795.805,A -85,B 0,C 180,E1 7382.935,E2 7382.935} C_VEL
LIN {X 0,Y 136.515,Z 789.523,A -85,B 0,C 180,E1 7376.599,E2 7376.599} C_VEL
LIN {X 0,Y 136.957,Z 781.216,A -85,B 0,C 180,E1 7369.908,E2 7369.908} C_VEL
LIN {X 0,Y 138.375,Z 770.81,A -85,B 0,C 180,E1 7363.2,E2 7363.2} C_VEL
LIN {X 0,Y 140.83,Z 758.932,A -85,B 0,C 180,E1 7357.015,E2 7357.015} C_VEL
LIN {X 0,Y 144.487,Z 744.559,A -85,B 0,C 180,E1 7351.026,E2 7351.026} C_VEL
LIN {X 0,Y 148.803,Z 729.031,A -85,B 0,C 180,E1 7345.87,E2 7345.87} C_VEL
LIN {X 0,Y 153.645,Z 711.76,A -85,B 0,C 180,E1 7341.337,E2 7341.337} C_VEL
LIN {X 0,Y 158.578,Z 693.19,A -85,B 0,C 180,E1 7337.536,E2 7337.536} C_VEL
LIN {X 0,Y 163.296,Z 673.628,A -85,B 0,C 180,E1 7334.433,E2 7334.433} C_VEL
LIN {X 0,Y 167.487,Z 653.476,A -85,B 0,C 180,E1 7331.991,E2 7331.991} C_VEL
LIN {X 0,Y 171.166,Z 631.549,A -85,B 0,C 180,E1 7330.053,E2 7330.053} C_VEL
LIN {X 0,Y 189.178,Z 504.226,A -85,B 0,C 180,E1 7322.443,E2 7322.443} C_VEL
LIN {X 0,Y 179.11,Z 481.792,A -85,B 0,C 180,E1 7318.055,E2 7318.055} C_VEL
LIN {X 0,Y 169.454,Z 462.099,A -85,B 0,C 180,E1 7313.379,E2 7313.379} C_VEL
LIN {X 0,Y 160.372,Z 445.3,A -85,B 0,C 180,E1 7308.484,E2 7308.484} C_VEL
LIN {X 0,Y 152.498,Z 432.233,A -85,B 0,C 180,E1 7303.749,E2 7303.749} C_VEL
LIN {X 0,Y 147.2,Z 423.69,A -85,B 0,C 180,E1 7299.962,E2 7299.962} C_VEL
LIN {X 0,Y 144.57,Z 418.952,A -85,B 0,C 180,E1 7297.151,E2 7297.151} C_VEL
LIN {X 0,Y 142.532,Z 415.103,A -85,B 0,C 180,E1 7294.829,E2 7294.829} C_VEL
LIN {X 0,Y 140.002,Z 411.467,A -85,B 0,C 180,E1 7292.046,E2 7292.046} C_VEL
LIN {X 0,Y 139.46,Z 409.427,A -85,B 0,C 180,E1 7290.924,E2 7290.924} C_VEL
LIN {X 0,Y 139.466,Z 409.422,A -85,B 0,C 180,E1 7284.24,E2 7284.24} C_VEL
LIN {X 0,Y 139.485,Z 409.559,A -85,B 0,C 180,E1 7277.772,E2 7277.772} C_VEL
LIN {X 0,Y 142.198,Z 417.038,A -85,B 0,C 180,E1 7271.978,E2 7271.978} C_VEL
LIN {X 0,Y 145.04,Z 425.148,A -85,B 0,C 180,E1 7266.432,E2 7266.432} C_VEL
LIN {X 0,Y 148.119,Z 435.119,A -85,B 0,C 180,E1 7260.476,E2 7260.476} C_VEL
LIN {X 0,Y 151.24,Z 446.63,A -85,B 0,C 180,E1 7254.407,E2 7254.407} C_VEL
LIN {X 0,Y 154.197,Z 458.956,A -85,B 0,C 180,E1 7248.593,E2 7248.593} C_VEL
LIN {X 0,Y 157.138,Z 472.827,A -85,B 0,C 180,E1 7242.686,E2 7242.686} C_VEL
LIN {X 0,Y 156.525,Z 475.073,A -85,B 0,C 180,E1 7242.057,E2 7242.057} C_VEL
LIN {X 0,Y 156.517,Z 503.478,A -85,B 0,C 180,E1 7239.45,E2 7239.45} C_VEL
LIN {X 0,Y 157.375,Z 527.732,A -85,B 0,C 180,E1 7237.141,E2 7237.141} C_VEL
LIN {X 0,Y 148.232,Z 621.833,A -85,B 0,C 180,E1 7229.253,E2 7229.253} C_VEL
LIN {X 0,Y 146.277,Z 641.754,A -85,B 0,C 180,E1 7226.817,E2 7226.817} C_VEL
LIN {X 0,Y 144.039,Z 660.87,A -85,B 0,C 180,E1 7223.609,E2 7223.609} C_VEL
LIN {X 0,Y 141.964,Z 678.536,A -85,B 0,C 180,E1 7219.76,E2 7219.76} C_VEL
LIN {X 0,Y 140.184,Z 694.683,A -85,B 0,C 180,E1 7215.302,E2 7215.302} C_VEL
LIN {X 0,Y 138.957,Z 709.49,A -85,B 0,C 180,E1 7210.154,E2 7210.154} C_VEL
LIN {X 0,Y 138.502,Z 721.695,A -85,B 0,C 180,E1 7204.97,E2 7204.97} C_VEL
LIN {X 0,Y 139.024,Z 733.929,A -85,B 0,C 180,E1 7198.579,E2 7198.579} C_VEL
LIN {X 0,Y 140.894,Z 743.672,A -85,B 0,C 180,E1 7192.251,E2 7192.251} C_VEL
LIN {X 0,Y 144.744,Z 752.118,A -85,B 0,C 180,E1 7185.601,E2 7185.601} C_VEL
LIN {X 0,Y 150.568,Z 758.44,A -85,B 0,C 180,E1 7179.394,E2 7179.394} C_VEL
LIN {X 0,Y 158.781,Z 763.197,A -85,B 0,C 180,E1 7173.443,E2 7173.443} C_VEL
LIN {X 0,Y 168.866,Z 766.012,A -85,B 0,C 180,E1 7168.199,E2 7168.199} C_VEL
LIN {X 0,Y 181.251,Z 767.078,A -85,B 0,C 180,E1 7163.433,E2 7163.433} C_VEL
LIN {X 0,Y 183.047,Z 767.157,A -85,B 0,C 180,E1 7162.763,E2 7162.763} C_VEL
LIN {X 0,Y 167.563,Z 772.542,A -85,B 0,C 180,E1 7157.219,E2 7157.219} C_VEL
LIN {X 0,Y 154.237,Z 776.739,A -85,B 0,C 180,E1 7149.925,E2 7149.925} C_VEL
LIN {X 0,Y 144.715,Z 779.393,A -85,B 0,C 180,E1 7141.049,E2 7141.049} C_VEL
LIN {X 0,Y 140.08,Z 780.301,A -85,B 0,C 180,E1 7131.348,E2 7131.348} C_VEL
LIN {X 0,Y 139.904,Z 780.375,A -85,B 0,C 180,E1 7130.499,E2 7130.499} C_VEL
LIN {X 0,Y 138.742,Z 785.669,A -85,B 0,C 180,E1 7127.465,E2 7127.465} C_VEL
LIN {X 0,Y 137.292,Z 789.782,A -85,B 0,C 180,E1 7124.801,E2 7124.801} C_VEL
LIN {X 0,Y 133.318,Z 795.075,A -85,B 0,C 180,E1 7120.397,E2 7120.397} C_VEL
LIN {X 0,Y 130.584,Z 799.371,A -85,B 0,C 180,E1 7116.028,E2 7116.028} C_VEL
LIN {X 0,Y 130.38,Z 801.125,A -85,B 0,C 180,E1 7114.213,E2 7114.213} C_VEL
LIN {X 0,Y 130.601,Z 805.268,A -85,B 0,C 180,E1 7109.561,E2 7109.561} C_VEL
LIN {X 0,Y 129.96,Z 808.433,A -85,B 0,C 180,E1 7104.703,E2 7104.703} C_VEL
LIN {X 0,Y 129.595,Z 812.229,A -85,B 0,C 180,E1 7096.162,E2 7096.162} C_VEL
LIN {X 0,Y 132.429,Z 814.785,A -85,B 0,C 180,E1 7086.412,E2 7086.412} C_VEL
LIN {X 0,Y 139.915,Z 815.716,A -85,B 0,C 180,E1 7076.615,E2 7076.615} C_VEL
LIN {X 0,Y 152.137,Z 814.917,A -85,B 0,C 180,E1 7067.905,E2 7067.905} C_VEL
LIN {X 0,Y 163.914,Z 813.177,A -85,B 0,C 180,E1 7062.431,E2 7062.431} C_VEL
LIN {X 0,Y 149.5,Z 812.096,A -85,B 0,C 180,E1 7055.111,E2 7055.111} C_VEL
LIN {X 0,Y 139.187,Z 809.385,A -85,B 0,C 180,E1 7046.908,E2 7046.908} C_VEL
LIN {X 0,Y 132.418,Z 804.871,A -85,B 0,C 180,E1 7037.579,E2 7037.579} C_VEL
LIN {X 0,Y 129.467,Z 799.245,A -85,B 0,C 180,E1 7028.885,E2 7028.885} C_VEL
LIN {X 0,Y 128.681,Z 792.977,A -85,B 0,C 180,E1 7021.335,E2 7021.335} C_VEL
LIN {X 0,Y 128.659,Z 786.018,A -85,B 0,C 180,E1 7014.648,E2 7014.648} C_VEL
LIN {X 0,Y 129.397,Z 776.748,A -85,B 0,C 180,E1 7007.504,E2 7007.504} C_VEL
LIN {X 0,Y 131.31,Z 765.277,A -85,B 0,C 180,E1 7000.425,E2 7000.425} C_VEL
LIN {X 0,Y 134.375,Z 752.206,A -85,B 0,C 180,E1 6993.959,E2 6993.959} C_VEL
LIN {X 0,Y 138.557,Z 737.003,A -85,B 0,C 180,E1 6987.967,E2 6987.967} C_VEL
LIN {X 0,Y 143.3,Z 720.612,A -85,B 0,C 180,E1 6982.875,E2 6982.875} C_VEL
LIN {X 0,Y 148.248,Z 703.151,A -85,B 0,C 180,E1 6978.626,E2 6978.626} C_VEL
LIN {X 0,Y 153.256,Z 684.147,A -85,B 0,C 180,E1 6975.031,E2 6975.031} C_VEL
LIN {X 0,Y 157.85,Z 664.575,A -85,B 0,C 180,E1 6972.174,E2 6972.174} C_VEL
LIN {X 0,Y 161.96,Z 643.716,A -85,B 0,C 180,E1 6969.892,E2 6969.892} C_VEL
LIN {X 0,Y 165.678,Z 619.503,A -85,B 0,C 180,E1 6968.009,E2 6968.009} C_VEL
LIN {X 0,Y 182.32,Z 506.499,A -85,B 0,C 180,E1 6961.12,E2 6961.12} C_VEL
LIN {X 0,Y 172.425,Z 484.265,A -85,B 0,C 180,E1 6956.52,E2 6956.52} C_VEL
LIN {X 0,Y 163.316,Z 465.549,A -85,B 0,C 180,E1 6951.835,E2 6951.835} C_VEL
LIN {X 0,Y 155.034,Z 450.067,A -85,B 0,C 180,E1 6947.064,E2 6947.064} C_VEL
LIN {X 0,Y 147.627,Z 437.504,A -85,B 0,C 180,E1 6942.319,E2 6942.319} C_VEL
LIN {X 0,Y 142.248,Z 429.11,A -85,B 0,C 180,E1 6938.488,E2 6938.488} C_VEL
LIN {X 0,Y 139.882,Z 425.27,A -85,B 0,C 180,E1 6936.567,E2 6936.567} C_VEL
LIN {X 0,Y 137.126,Z 420.431,A -85,B 0,C 180,E1 6933.344,E2 6933.344} C_VEL
LIN {X 0,Y 134.994,Z 416.869,A -85,B 0,C 180,E1 6930.735,E2 6930.735} C_VEL
LIN {X 0,Y 134.533,Z 415.707,A -85,B 0,C 180,E1 6930,E2 6930} C_VEL
LIN {X 0,Y 132.08,Z 412.508,A -85,B 0,C 180,E1 6926.962,E2 6926.962} C_VEL
LIN {X 0,Y 131.521,Z 410.41,A -85,B 0,C 180,E1 6925.64,E2 6925.64} C_VEL
LIN {X 0,Y 131.552,Z 410.593,A -85,B 0,C 180,E1 6921.477,E2 6921.477} C_VEL
LIN {X 0,Y 133.362,Z 415.672,A -85,B 0,C 180,E1 6917.002,E2 6917.002} C_VEL
LIN {X 0,Y 135.541,Z 421.374,A -85,B 0,C 180,E1 6912.395,E2 6912.395} C_VEL
LIN {X 0,Y 138.314,Z 429.604,A -85,B 0,C 180,E1 6906.572,E2 6906.572} C_VEL
LIN {X 0,Y 141.237,Z 439.355,A -85,B 0,C 180,E1 6900.548,E2 6900.548} C_VEL
LIN {X 0,Y 144.21,Z 450.687,A -85,B 0,C 180,E1 6894.38,E2 6894.38} C_VEL
LIN {X 0,Y 147.02,Z 462.94,A -85,B 0,C 180,E1 6888.426,E2 6888.426} C_VEL
LIN {X 0,Y 149.281,Z 474.403,A -85,B 0,C 180,E1 6883.357,E2 6883.357} C_VEL
LIN {X 0,Y 148.97,Z 502.003,A -85,B 0,C 180,E1 6880.691,E2 6880.691} C_VEL
LIN {X 0,Y 149.761,Z 527.993,A -85,B 0,C 180,E1 6878.078,E2 6878.078} C_VEL
LIN {X 0,Y 140.568,Z 619.079,A -85,B 0,C 180,E1 6870.054,E2 6870.054} C_VEL
LIN {X 0,Y 138.704,Z 638.208,A -85,B 0,C 180,E1 6867.708,E2 6867.708} C_VEL
LIN {X 0,Y 136.55,Z 656.607,A -85,B 0,C 180,E1 6864.669,E2 6864.669} C_VEL
LIN {X 0,Y 134.46,Z 674.096,A -85,B 0,C 180,E1 6860.913,E2 6860.913} C_VEL
LIN {X 0,Y 132.506,Z 691.136,A -85,B 0,C 180,E1 6856.213,E2 6856.213} C_VEL
LIN {X 0,Y 131.12,Z 706.845,A -85,B 0,C 180,E1 6850.768,E2 6850.768} C_VEL
LIN {X 0,Y 130.583,Z 720.479,A -85,B 0,C 180,E1 6844.832,E2 6844.832} C_VEL
LIN {X 0,Y 131.004,Z 731.609,A -85,B 0,C 180,E1 6838.957,E2 6838.957} C_VEL
LIN {X 0,Y 132.83,Z 742.102,A -85,B 0,C 180,E1 6832.213,E2 6832.213} C_VEL
LIN {X 0,Y 136.427,Z 750.733,A -85,B 0,C 180,E1 6825.571,E2 6825.571} C_VEL
LIN {X 0,Y 142.28,Z 757.803,A -85,B 0,C 180,E1 6818.999,E2 6818.999} C_VEL
LIN {X 0,Y 150.625,Z 763.343,A -85,B 0,C 180,E1 6812.741,E2 6812.741} C_VEL
LIN {X 0,Y 160.928,Z 766.939,A -85,B 0,C 180,E1 6807.28,E2 6807.28} C_VEL
LIN {X 0,Y 171.825,Z 768.762,A -85,B 0,C 180,E1 6802.865,E2 6802.865} C_VEL
LIN {X 0,Y 155.918,Z 773.2,A -85,B 0,C 180,E1 6796.439,E2 6796.439} C_VEL
LIN {X 0,Y 143.4,Z 776.206,A -85,B 0,C 180,E1 6788.357,E2 6788.357} C_VEL
LIN {X 0,Y 135.196,Z 777.701,A -85,B 0,C 180,E1 6778.732,E2 6778.732} C_VEL
LIN {X 0,Y 132.385,Z 777.893,A -85,B 0,C 180,E1 6771.14,E2 6771.14} C_VEL
LIN {X 0,Y 130.62,Z 786.379,A -85,B 0,C 180,E1 6765.996,E2 6765.996} C_VEL
LIN {X 0,Y 130.108,Z 795.52,A -85,B 0,C 180,E1 6759.287,E2 6759.287} C_VEL
LIN {X 0,Y 130.38,Z 801.125,A -85,B 0,C 180,E1 6754.213,E2 6754.213} C_VEL
LIN {X 0,Y 129.923,Z 803.113,A -85,B 0,C 180,E1 6751.954,E2 6751.954} C_VEL
LIN {X 0,Y 127.614,Z 805.28,A -85,B 0,C 180,E1 6748.512,E2 6748.512} C_VEL
LIN {X 0,Y 122.07,Z 808.365,A -85,B 0,C 180,E1 6740.603,E2 6740.603} C_VEL
LIN {X 0,Y 121.768,Z 809.06,A -85,B 0,C 180,E1 6738.747,E2 6738.747} C_VEL
LIN {X 0,Y 123.676,Z 812.59,A -85,B 0,C 180,E1 6728.168,E2 6728.168} C_VEL
LIN {X 0,Y 130.545,Z 814.472,A -85,B 0,C 180,E1 6717.404,E2 6717.404} C_VEL
LIN {X 0,Y 142.21,Z 814.6,A -85,B 0,C 180,E1 6708.092,E2 6708.092} C_VEL
LIN {X 0,Y 153.249,Z 813.674,A -85,B 0,C 180,E1 6702.317,E2 6702.317} C_VEL
LIN {X 0,Y 139.331,Z 811.536,A -85,B 0,C 180,E1 6694.535,E2 6694.535} C_VEL
LIN {X 0,Y 129.118,Z 807.623,A -85,B 0,C 180,E1 6685.207,E2 6685.207} C_VEL
LIN {X 0,Y 123.216,Z 801.964,A -85,B 0,C 180,E1 6675.05,E2 6675.05} C_VEL
LIN {X 0,Y 121.081,Z 795.243,A -85,B 0,C 180,E1 6665.686,E2 6665.686} C_VEL
LIN {X 0,Y 120.723,Z 788.758,A -85,B 0,C 180,E1 6658.576,E2 6658.576} C_VEL
LIN {X 0,Y 120.975,Z 780.754,A -85,B 0,C 180,E1 6651.444,E2 6651.444} C_VEL
LIN {X 0,Y 122.144,Z 770.944,A -85,B 0,C 180,E1 6644.327,E2 6644.327} C_VEL
LIN {X 0,Y 124.548,Z 759.057,A -85,B 0,C 180,E1 6637.335,E2 6637.335} C_VEL
LIN {X 0,Y 128.307,Z 744.703,A -85,B 0,C 180,E1 6630.597,E2 6630.597} C_VEL
LIN {X 0,Y 132.85,Z 729.167,A -85,B 0,C 180,E1 6624.847,E2 6624.847} C_VEL
LIN {X 0,Y 137.992,Z 711.889,A -85,B 0,C 180,E1 6619.843,E2 6619.843} C_VEL
LIN {X 0,Y 143.216,Z 693.466,A -85,B 0,C 180,E1 6615.721,E2 6615.721} C_VEL
LIN {X 0,Y 148.487,Z 673.034,A -85,B 0,C 180,E1 6612.208,E2 6612.208} C_VEL
LIN {X 0,Y 153.038,Z 652.378,A -85,B 0,C 180,E1 6609.561,E2 6609.561} C_VEL
LIN {X 0,Y 156.998,Z 630.062,A -85,B 0,C 180,E1 6607.486,E2 6607.486} C_VEL
LIN {X 0,Y 175.48,Z 508.747,A -85,B 0,C 180,E1 6599.717,E2 6599.717} C_VEL
LIN {X 0,Y 165.908,Z 486.957,A -85,B 0,C 180,E1 6594.952,E2 6594.952} C_VEL
LIN {X 0,Y 156.602,Z 467.726,A -85,B 0,C 180,E1 6589.828,E2 6589.828} C_VEL
LIN {X 0,Y 148.315,Z 452.168,A -85,B 0,C 180,E1 6584.644,E2 6584.644} C_VEL
LIN {X 0,Y 141.074,Z 439.944,A -85,B 0,C 180,E1 6579.567,E2 6579.567} C_VEL
LIN {X 0,Y 135.426,Z 431.148,A -85,B 0,C 180,E1 6575.083,E2 6575.083} C_VEL
LIN {X 0,Y 132.169,Z 426.305,A -85,B 0,C 180,E1 6572.168,E2 6572.168} C_VEL
LIN {X 0,Y 129.927,Z 422.096,A -85,B 0,C 180,E1 6569.118,E2 6569.118} C_VEL
LIN {X 0,Y 127.564,Z 418.707,A -85,B 0,C 180,E1 6565.955,E2 6565.955} C_VEL
LIN {X 0,Y 126.797,Z 416.87,A -85,B 0,C 180,E1 6564.57,E2 6564.57} C_VEL
LIN {X 0,Y 125.111,Z 415.178,A -85,B 0,C 180,E1 6562.076,E2 6562.076} C_VEL
LIN {X 0,Y 127.747,Z 422.423,A -85,B 0,C 180,E1 6555.495,E2 6555.495} C_VEL
LIN {X 0,Y 130.531,Z 430.543,A -85,B 0,C 180,E1 6549.152,E2 6549.152} C_VEL
LIN {X 0,Y 133.163,Z 439.349,A -85,B 0,C 180,E1 6543.223,E2 6543.223} C_VEL
LIN {X 0,Y 135.745,Z 449.008,A -85,B 0,C 180,E1 6537.473,E2 6537.473} C_VEL
LIN {X 0,Y 138.521,Z 460.775,A -85,B 0,C 180,E1 6531.221,E2 6531.221} C_VEL
LIN {X 0,Y 141.184,Z 473.648,A -85,B 0,C 180,E1 6525.089,E2 6525.089} C_VEL
LIN {X 0,Y 141.587,Z 475.26,A -85,B 0,C 180,E1 6524.608,E2 6524.608} C_VEL
LIN {X 0,Y 141.691,Z 479.265,A -85,B 0,C 180,E1 6524.175,E2 6524.175} C_VEL
LIN {X 0,Y 141.697,Z 510.677,A -85,B 0,C 180,E1 6520.952,E2 6520.952} C_VEL
LIN {X 0,Y 142.151,Z 528.441,A -85,B 0,C 180,E1 6519.081,E2 6519.081} C_VEL
LIN {X 0,Y 132.287,Z 623.32,A -85,B 0,C 180,E1 6510.134,E2 6510.134} C_VEL
LIN {X 0,Y 130.23,Z 642.815,A -85,B 0,C 180,E1 6507.43,E2 6507.43} C_VEL
LIN {X 0,Y 127.907,Z 661.796,A -85,B 0,C 180,E1 6503.85,E2 6503.85} C_VEL
LIN {X 0,Y 125.67,Z 680.313,A -85,B 0,C 180,E1 6499.28,E2 6499.28} C_VEL
LIN {X 0,Y 123.956,Z 696.27,A -85,B 0,C 180,E1 6494.243,E2 6494.243} C_VEL
LIN {X 0,Y 122.919,Z 710.513,A -85,B 0,C 180,E1 6488.656,E2 6488.656} C_VEL
LIN {X 0,Y 122.714,Z 722.781,A -85,B 0,C 180,E1 6482.803,E2 6482.803} C_VEL
LIN {X 0,Y 123.569,Z 734.071,A -85,B 0,C 180,E1 6476.289,E2 6476.289} C_VEL
LIN {X 0,Y 126.13,Z 744.562,A -85,B 0,C 180,E1 6469.033,E2 6469.033} C_VEL
LIN {X 0,Y 130.963,Z 753.365,A -85,B 0,C 180,E1 6461.759,E2 6461.759} C_VEL
LIN {X 0,Y 138.446,Z 760.573,A -85,B 0,C 180,E1 6454.78,E2 6454.78} C_VEL
LIN {X 0,Y 148.1,Z 765.772,A -85,B 0,C 180,E1 6448.679,E2 6448.679} C_VEL
LIN {X 0,Y 159.608,Z 769.17,A -85,B 0,C 180,E1 6443.479,E2 6443.479} C_VEL
LIN {X 0,Y 160.72,Z 769.479,A -85,B 0,C 180,E1 6442.927,E2 6442.927} C_VEL
LIN {X 0,Y 145.075,Z 772.846,A -85,B 0,C 180,E1 6435.789,E2 6435.789} C_VEL
LIN {X 0,Y 133.305,Z 774.807,A -85,B 0,C 180,E1 6426.873,E2 6426.873} C_VEL
LIN {X 0,Y 126.279,Z 775.283,A -85,B 0,C 180,E1 6416.321,E2 6416.321} C_VEL
LIN {X 0,Y 125.006,Z 775.131,A -85,B 0,C 180,E1 6411.958,E2 6411.958} C_VEL
LIN {X 0,Y 122.994,Z 782.993,A -85,B 0,C 180,E1 6407.017,E2 6407.017} C_VEL
LIN {X 0,Y 122.342,Z 792.619,A -85,B 0,C 180,E1 6399.882,E2 6399.882} C_VEL
LIN {X 0,Y 122.699,Z 799.777,A -85,B 0,C 180,E1 6393.27,E2 6393.27} C_VEL
LIN {X 0,Y 122.861,Z 803.696,A -85,B 0,C 180,E1 6388.601,E2 6388.601} C_VEL
LIN {X 0,Y 122.008,Z 807.328,A -85,B 0,C 180,E1 6382.466,E2 6382.466} C_VEL
LIN {X 0,Y 121.768,Z 809.06,A -85,B 0,C 180,E1 6378.747,E2 6378.747} C_VEL
LIN {X 0,Y 121.011,Z 810.174,A -85,B 0,C 180,E1 6375.138,E2 6375.138} C_VEL
LIN {X 0,Y 117.853,Z 811.516,A -85,B 0,C 180,E1 6364.779,E2 6364.779} C_VEL
LIN {X 0,Y 118.83,Z 811.966,A -85,B 0,C 180,E1 6361.863,E2 6361.863} C_VEL
LIN {X 0,Y 128.235,Z 813.541,A -85,B 0,C 180,E1 6351.408,E2 6351.408} C_VEL
LIN {X 0,Y 142.909,Z 813.517,A -85,B 0,C 180,E1 6342.33,E2 6342.33} C_VEL
LIN {X 0,Y 129.218,Z 810.33,A -85,B 0,C 180,E1 6333.856,E2 6333.856} C_VEL
LIN {X 0,Y 119.558,Z 805.335,A -85,B 0,C 180,E1 6323.666,E2 6323.666} C_VEL
LIN {X 0,Y 114.59,Z 798.929,A -85,B 0,C 180,E1 6313.112,E2 6313.112} C_VEL
LIN {X 0,Y 113.082,Z 792.116,A -85,B 0,C 180,E1 6304.056,E2 6304.056} C_VEL
LIN {X 0,Y 112.864,Z 784.892,A -85,B 0,C 180,E1 6296.444,E2 6296.444} C_VEL
LIN {X 0,Y 113.389,Z 776.008,A -85,B 0,C 180,E1 6288.813,E2 6288.813} C_VEL
LIN {X 0,Y 115.224,Z 764.389,A -85,B 0,C 180,E1 6280.746,E2 6280.746} C_VEL
LIN {X 0,Y 118.403,Z 751.139,A -85,B 0,C 180,E1 6273.412,E2 6273.412} C_VEL
LIN {X 0,Y 122.691,Z 736.292,A -85,B 0,C 180,E1 6266.905,E2 6266.905} C_VEL
LIN {X 0,Y 127.774,Z 719.707,A -85,B 0,C 180,E1 6261.242,E2 6261.242} C_VEL
LIN {X 0,Y 133.094,Z 702.053,A -85,B 0,C 180,E1 6256.575,E2 6256.575} C_VEL
LIN {X 0,Y 138.569,Z 682.558,A -85,B 0,C 180,E1 6252.608,E2 6252.608} C_VEL
LIN {X 0,Y 143.523,Z 662.584,A -85,B 0,C 180,E1 6249.539,E2 6249.539} C_VEL
LIN {X 0,Y 148.079,Z 640.34,A -85,B 0,C 180,E1 6247.037,E2 6247.037} C_VEL
LIN {X 0,Y 152.841,Z 610.332,A -85,B 0,C 180,E1 6244.674,E2 6244.674} C_VEL
LIN {X 0,Y 168.715,Z 511.102,A -85,B 0,C 180,E1 6238.253,E2 6238.253} C_VEL
LIN {X 0,Y 159.72,Z 490.334,A -85,B 0,C 180,E1 6233.472,E2 6233.472} C_VEL
LIN {X 0,Y 150.805,Z 471.615,A -85,B 0,C 180,E1 6228.207,E2 6228.207} C_VEL
LIN {X 0,Y 143.058,Z 456.884,A -85,B 0,C 180,E1 6223.027,E2 6223.027} C_VEL
LIN {X 0,Y 136.653,Z 445.777,A -85,B 0,C 180,E1 6218.203,E2 6218.203} C_VEL
LIN {X 0,Y 131.244,Z 437.164,A -85,B 0,C 180,E1 6213.615,E2 6213.615} C_VEL
LIN {X 0,Y 128.22,Z 432.607,A -85,B 0,C 180,E1 6210.782,E2 6210.782} C_VEL
LIN {X 0,Y 125.281,Z 428.199,A -85,B 0,C 180,E1 6207.713,E2 6207.713} C_VEL
LIN {X 0,Y 122.887,Z 424.29,A -85,B 0,C 180,E1 6204.397,E2 6204.397} C_VEL
LIN {X 0,Y 121.919,Z 422.931,A -85,B 0,C 180,E1 6202.901,E2 6202.901} C_VEL
LIN {X 0,Y 119.485,Z 422.419,A -85,B 0,C 180,E1 6200.122,E2 6200.122} C_VEL
LIN {X 0,Y 122.042,Z 429.339,A -85,B 0,C 180,E1 6193.826,E2 6193.826} C_VEL
LIN {X 0,Y 124.704,Z 437.948,A -85,B 0,C 180,E1 6187.23,E2 6187.23} C_VEL
LIN {X 0,Y 127.35,Z 447.489,A -85,B 0,C 180,E1 6180.871,E2 6180.871} C_VEL
LIN {X 0,Y 130.061,Z 458.82,A -85,B 0,C 180,E1 6174.249,E2 6174.249} C_VEL
LIN {X 0,Y 132.656,Z 471.105,A -85,B 0,C 180,E1 6167.87,E2 6167.87} C_VEL
LIN {X 0,Y 133.422,Z 474.772,A -85,B 0,C 180,E1 6166.228,E2 6166.228} C_VEL
LIN {X 0,Y 134.417,Z 478.55,A -85,B 0,C 180,E1 6165.61,E2 6165.61} C_VEL
LIN {X 0,Y 134.147,Z 509.381,A -85,B 0,C 180,E1 6162.296,E2 6162.296} C_VEL
LIN {X 0,Y 134.543,Z 528.692,A -85,B 0,C 180,E1 6160.137,E2 6160.137} C_VEL
LIN {X 0,Y 124.607,Z 620.727,A -85,B 0,C 180,E1 6150.968,E2 6150.968} C_VEL
LIN {X 0,Y 122.552,Z 640.241,A -85,B 0,C 180,E1 6148.219,E2 6148.219} C_VEL
LIN {X 0,Y 120.329,Z 658.229,A -85,B 0,C 180,E1 6144.811,E2 6144.811} C_VEL
LIN {X 0,Y 118.203,Z 675.498,A -85,B 0,C 180,E1 6140.552,E2 6140.552} C_VEL
LIN {X 0,Y 116.288,Z 692.469,A -85,B 0,C 180,E1 6135.204,E2 6135.204} C_VEL
LIN {X 0,Y 115.11,Z 707.487,A -85,B 0,C 180,E1 6129.248,E2 6129.248} C_VEL
LIN {X 0,Y 114.83,Z 720.385,A -85,B 0,C 180,E1 6122.995,E2 6122.995} C_VEL
LIN {X 0,Y 115.688,Z 732.212,A -85,B 0,C 180,E1 6116.036,E2 6116.036} C_VEL
LIN {X 0,Y 118.117,Z 742.649,A -85,B 0,C 180,E1 6108.774,E2 6108.774} C_VEL
LIN {X 0,Y 122.691,Z 751.618,A -85,B 0,C 180,E1 6101.469,E2 6101.469} C_VEL
LIN {X 0,Y 129.767,Z 759.228,A -85,B 0,C 180,E1 6094.439,E2 6094.439} C_VEL
LIN {X 0,Y 138.903,Z 765.064,A -85,B 0,C 180,E1 6088.3,E2 6088.3} C_VEL
LIN {X 0,Y 149.809,Z 769.31,A -85,B 0,C 180,E1 6082.947,E2 6082.947} C_VEL
LIN {X 0,Y 134.433,Z 771.651,A -85,B 0,C 180,E1 6074.957,E2 6074.957} C_VEL
LIN {X 0,Y 123.548,Z 772.61,A -85,B 0,C 180,E1 6065.072,E2 6065.072} C_VEL
LIN {X 0,Y 117.742,Z 772.14,A -85,B 0,C 180,E1 6052.862,E2 6052.862} C_VEL
LIN {X 0,Y 115.432,Z 779.457,A -85,B 0,C 180,E1 6048.17,E2 6048.17} C_VEL
LIN {X 0,Y 114.597,Z 789.573,A -85,B 0,C 180,E1 6040.558,E2 6040.558} C_VEL
LIN {X 0,Y 114.952,Z 797.078,A -85,B 0,C 180,E1 6033.491,E2 6033.491} C_VEL
LIN {X 0,Y 115.244,Z 800.919,A -85,B 0,C 180,E1 6029.006,E2 6029.006} C_VEL
LIN {X 0,Y 114.515,Z 804.347,A -85,B 0,C 180,E1 6023.483,E2 6023.483} C_VEL
LIN {X 0,Y 114.522,Z 808.773,A -85,B 0,C 180,E1 6013.255,E2 6013.255} C_VEL
LIN {X 0,Y 118.83,Z 811.966,A -85,B 0,C 180,E1 6001.863,E2 6001.863} C_VEL
LIN {X 0,Y 120.365,Z 812.442,A -85,B 0,C 180,E1 5998.22,E2 5998.22} C_VEL
LIN {X 0,Y 123.657,Z 812.489,A -85,B 0,C 180,E1 5988.622,E2 5988.622} C_VEL
LIN {X 0,Y 126.877,Z 812.523,A -85,B 0,C 180,E1 5985.679,E2 5985.679} C_VEL
LIN {X 0,Y 132.523,Z 812.629,A -85,B 0,C 180,E1 5982.283,E2 5982.283} C_VEL
LIN {X 0,Y 119.185,Z 808.431,A -85,B 0,C 180,E1 5973.044,E2 5973.044} C_VEL
LIN {X 0,Y 110.444,Z 802.693,A -85,B 0,C 180,E1 5962.347,E2 5962.347} C_VEL
LIN {X 0,Y 106.251,Z 795.714,A -85,B 0,C 180,E1 5951.397,E2 5951.397} C_VEL
LIN {X 0,Y 105.181,Z 788.98,A -85,B 0,C 180,E1 5942.724,E2 5942.724} C_VEL
LIN {X 0,Y 105.055,Z 781.657,A -85,B 0,C 180,E1 5935.086,E2 5935.086} C_VEL
LIN {X 0,Y 105.803,Z 772.082,A -85,B 0,C 180,E1 5926.89,E2 5926.89} C_VEL
LIN {X 0,Y 107.914,Z 760.445,A -85,B 0,C 180,E1 5918.816,E2 5918.816} C_VEL
LIN {X 0,Y 111.579,Z 746.384,A -85,B 0,C 180,E1 5911.059,E2 5911.059} C_VEL
LIN {X 0,Y 116.408,Z 730.562,A -85,B 0,C 180,E1 5904.262,E2 5904.262} C_VEL
LIN {X 0,Y 121.563,Z 714.366,A -85,B 0,C 180,E1 5898.852,E2 5898.852} C_VEL
LIN {X 0,Y 127.313,Z 695.567,A -85,B 0,C 180,E1 5894.06,E2 5894.06} C_VEL
LIN {X 0,Y 132.896,Z 675.68,A -85,B 0,C 180,E1 5890.212,E2 5890.212} C_VEL
LIN {X 0,Y 137.871,Z 655.165,A -85,B 0,C 180,E1 5887.257,E2 5887.257} C_VEL
LIN {X 0,Y 142.222,Z 632.958,A -85,B 0,C 180,E1 5884.953,E2 5884.953} C_VEL
LIN {X 0,Y 161.988,Z 513.393,A -85,B 0,C 180,E1 5876.682,E2 5876.682} C_VEL
LIN {X 0,Y 153.145,Z 492.744,A -85,B 0,C 180,E1 5871.647,E2 5871.647} C_VEL
LIN {X 0,Y 144.808,Z 474.959,A -85,B 0,C 180,E1 5866.307,E2 5866.307} C_VEL
LIN {X 0,Y 137.162,Z 460.189,A -85,B 0,C 180,E1 5860.766,E2 5860.766} C_VEL
LIN {X 0,Y 130.668,Z 448.794,A -85,B 0,C 180,E1 5855.379,E2 5855.379} C_VEL
LIN {X 0,Y 124.928,Z 439.648,A -85,B 0,C 180,E1 5849.897,E2 5849.897} C_VEL
LIN {X 0,Y 121.556,Z 434.665,A -85,B 0,C 180,E1 5846.227,E2 5846.227} C_VEL
LIN {X 0,Y 118.776,Z 430.342,A -85,B 0,C 180,E1 5842.746,E2 5842.746} C_VEL
LIN {X 0,Y 116.088,Z 430.195,A -85,B 0,C 180,E1 5840.081,E2 5840.081} C_VEL
LIN {X 0,Y 114.073,Z 429.908,A -85,B 0,C 180,E1 5837.824,E2 5837.824} C_VEL
LIN {X 0,Y 116.243,Z 436.465,A -85,B 0,C 180,E1 5831.962,E2 5831.962} C_VEL
LIN {X 0,Y 118.819,Z 445.472,A -85,B 0,C 180,E1 5825.118,E2 5825.118} C_VEL
LIN {X 0,Y 121.239,Z 455.21,A -85,B 0,C 180,E1 5818.697,E2 5818.697} C_VEL
